LIN {X 0,Y 337.999,Z 716.277,A -85,B 0,C 180,E1 -25443.497,E2 -25443.497} C_VEL
LIN {X 0,Y 342.458,Z 719.963,A -85,B 0,C 180,E1 -25446.093,E2 -25446.093} C_VEL
LIN {X 0,Y 346.569,Z 722.702,A -85,B 0,C 180,E1 -25448.688,E2 -25448.688} C_VEL
LIN {X 0,Y 349.968,Z 724.791,A -85,B 0,C 180,E1 -25450.993,E2 -25450.993} C_VEL
LIN {X 0,Y 353.266,Z 727.665,A -85,B 0,C 180,E1 -25453.67,E2 -25453.67} C_VEL
LIN {X 0,Y 355.856,Z 729.583,A -85,B 0,C 180,E1 -25456.067,E2 -25456.067} C_VEL
LIN {X 0,Y 358.314,Z 731.084,A -85,B 0,C 180,E1 -25458.723,E2 -25458.723} C_VEL
LIN {X 0,Y 360.355,Z 731.966,A -85,B 0,C 180,E1 -25461.416,E2 -25461.416} C_VEL
LIN {X 0,Y 361.794,Z 732.692,A -85,B 0,C 180,E1 -25464.054,E2 -25464.054} C_VEL
LIN {X 0,Y 362.724,Z 733.17,A -85,B 0,C 180,E1 -25466.668,E2 -25466.668} C_VEL
LIN {X 0,Y 363.106,Z 733.308,A -85,B 0,C 180,E1 -25468.891,E2 -25468.891} C_VEL
LIN {X 0,Y 363.106,Z 733.292,A -85,B 0,C 180,E1 -25471.109,E2 -25471.109} C_VEL
LIN {X 0,Y 362.712,Z 733.195,A -85,B 0,C 180,E1 -25473.332,E2 -25473.332} C_VEL
LIN {X 0,Y 361.809,Z 732.656,A -85,B 0,C 180,E1 -25475.946,E2 -25475.946} C_VEL
LIN {X 0,Y 360.322,Z 731.939,A -85,B 0,C 180,E1 -25478.61,E2 -25478.61} C_VEL
LIN {X 0,Y 358.3,Z 731.072,A -85,B 0,C 180,E1 -25481.312,E2 -25481.312} C_VEL
LIN {X 0,Y 355.654,Z 729.459,A -85,B 0,C 180,E1 -25484.125,E2 -25484.125} C_VEL
LIN {X 0,Y 352.777,Z 727.309,A -85,B 0,C 180,E1 -25486.738,E2 -25486.738} C_VEL
LIN {X 0,Y 349.188,Z 724.198,A -85,B 0,C 180,E1 -25489.587,E2 -25489.587} C_VEL
LIN {X 0,Y 344.756,Z 721.495,A -85,B 0,C 180,E1 -25492.513,E2 -25492.513} C_VEL
LIN {X 0,Y 340.447,Z 718.436,A -85,B 0,C 180,E1 -25495.072,E2 -25495.072} C_VEL
LIN {X 0,Y 336.743,Z 715.339,A -85,B 0,C 180,E1 -25497.172,E2 -25497.172} C_VEL
LIN {X 0,Y 332.718,Z 712.68,A -85,B 0,C 180,E1 -25499.253,E2 -25499.253} C_VEL
LIN {X 0,Y 327.18,Z 708.25,A -85,B 0,C 180,E1 -25501.98,E2 -25501.98} C_VEL
LIN {X 0,Y 322.544,Z 704.803,A -85,B 0,C 180,E1 -25504.108,E2 -25504.108} C_VEL
LIN {X 0,Y 316.501,Z 699.903,A -85,B 0,C 180,E1 -25506.755,E2 -25506.755} C_VEL
LIN {X 0,Y 309.747,Z 694.783,A -85,B 0,C 180,E1 -25509.517,E2 -25509.517} C_VEL
LIN {X 0,Y 303.112,Z 689.395,A -85,B 0,C 180,E1 -25512.103,E2 -25512.103} C_VEL
LIN {X 0,Y 296.74,Z 684.407,A -85,B 0,C 180,E1 -25514.411,E2 -25514.411} C_VEL
LIN {X 0,Y 289.825,Z 679.065,A -85,B 0,C 180,E1 -25516.73,E2 -25516.73} C_VEL
LIN {X 0,Y 282.712,Z 673.492,A -85,B 0,C 180,E1 -25518.913,E2 -25518.913} C_VEL
LIN {X 0,Y 268.912,Z 662.781,A -85,B 0,C 180,E1 -25522.994,E2 -25522.994} C_VEL
LIN {X 0,Y 252.75,Z 647.426,A -85,B 0,C 180,E1 -25529.042,E2 -25529.042} C_VEL
LIN {X 0,Y 243.109,Z 634.604,A -85,B 0,C 180,E1 -25533.946,E2 -25533.946} C_VEL
LIN {X 0,Y 236.411,Z 622.152,A -85,B 0,C 180,E1 -25538.53,E2 -25538.53} C_VEL
LIN {X 0,Y 233.122,Z 614.521,A -85,B 0,C 180,E1 -25541.432,E2 -25541.432} C_VEL
LIN {X 0,Y 229.896,Z 607.668,A -85,B 0,C 180,E1 -25544.826,E2 -25544.826} C_VEL
LIN {X 0,Y 227.317,Z 602.559,A -85,B 0,C 180,E1 -25548.255,E2 -25548.255} C_VEL
LIN {X 0,Y 225.85,Z 599.593,A -85,B 0,C 180,E1 -25550.824,E2 -25550.824} C_VEL
LIN {X 0,Y 224.425,Z 596.183,A -85,B 0,C 180,E1 -25554.61,E2 -25554.61} C_VEL
LIN {X 0,Y 223.643,Z 595.09,A -85,B 0,C 180,E1 -25560,E2 -25560} C_VEL
LIN {X 0,Y 224.47,Z 596.375,A -85,B 0,C 180,E1 -25565.165,E2 -25565.165} C_VEL
LIN {X 0,Y 226.423,Z 600.662,A -85,B 0,C 180,E1 -25569.83,E2 -25569.83} C_VEL
LIN {X 0,Y 228.163,Z 604.251,A -85,B 0,C 180,E1 -25572.565,E2 -25572.565} C_VEL
LIN {X 0,Y 230.141,Z 608.221,A -85,B 0,C 180,E1 -25575.05,E2 -25575.05} C_VEL
LIN {X 0,Y 232.646,Z 613.57,A -85,B 0,C 180,E1 -25577.702,E2 -25577.702} C_VEL
LIN {X 0,Y 234.172,Z 617.919,A -85,B 0,C 180,E1 -25579.22,E2 -25579.22} C_VEL
LIN {X 0,Y 228.253,Z 677.793,A -85,B 0,C 180,E1 -25580.525,E2 -25580.525} C_VEL
LIN {X 0,Y 225.904,Z 694.176,A -85,B 0,C 180,E1 -25580.947,E2 -25580.947} C_VEL
LIN {X 0,Y 222.958,Z 708.344,A -85,B 0,C 180,E1 -25581.432,E2 -25581.432} C_VEL
LIN {X 0,Y 219.343,Z 721.676,A -85,B 0,C 180,E1 -25582.002,E2 -25582.002} C_VEL
LIN {X 0,Y 215.576,Z 733.24,A -85,B 0,C 180,E1 -25582.632,E2 -25582.632} C_VEL
LIN {X 0,Y 210.564,Z 746.285,A -85,B 0,C 180,E1 -25583.53,E2 -25583.53} C_VEL
LIN {X 0,Y 204.879,Z 759,A -85,B 0,C 180,E1 -25584.631,E2 -25584.631} C_VEL
LIN {X 0,Y 199.091,Z 770.319,A -85,B 0,C 180,E1 -25585.824,E2 -25585.824} C_VEL
LIN {X 0,Y 192.723,Z 781.446,A -85,B 0,C 180,E1 -25587.27,E2 -25587.27} C_VEL
LIN {X 0,Y 185.768,Z 792.275,A -85,B 0,C 180,E1 -25588.973,E2 -25588.973} C_VEL
LIN {X 0,Y 179.725,Z 800.954,A -85,B 0,C 180,E1 -25590.653,E2 -25590.653} C_VEL
LIN {X 0,Y 173.216,Z 809.59,A -85,B 0,C 180,E1 -25592.661,E2 -25592.661} C_VEL
LIN {X 0,Y 164.386,Z 820.104,A -85,B 0,C 180,E1 -25595.68,E2 -25595.68} C_VEL
LIN {X 0,Y 157.519,Z 827.783,A -85,B 0,C 180,E1 -25598.491,E2 -25598.491} C_VEL
LIN {X 0,Y 150.758,Z 834.958,A -85,B 0,C 180,E1 -25601.766,E2 -25601.766} C_VEL
LIN {X 0,Y 144.568,Z 841.096,A -85,B 0,C 180,E1 -25605.18,E2 -25605.18} C_VEL
LIN {X 0,Y 137.225,Z 848.046,A -85,B 0,C 180,E1 -25610.195,E2 -25610.195} C_VEL
LIN {X 0,Y 131.064,Z 853.813,A -85,B 0,C 180,E1 -25615.735,E2 -25615.735} C_VEL
LIN {X 0,Y 127.275,Z 857.437,A -85,B 0,C 180,E1 -25620.201,E2 -25620.201} C_VEL
LIN {X 0,Y 123.381,Z 861.307,A -85,B 0,C 180,E1 -25626.502,E2 -25626.502} C_VEL
LIN {X 0,Y 120.659,Z 864.176,A -85,B 0,C 180,E1 -25633.069,E2 -25633.069} C_VEL
LIN {X 0,Y 119.367,Z 866.085,A -85,B 0,C 180,E1 -25639.827,E2 -25639.827} C_VEL
LIN {X 0,Y 119.17,Z 866.774,A -85,B 0,C 180,E1 -25643.226,E2 -25643.226} C_VEL
LIN {X 0,Y 119.331,Z 867.267,A -85,B 0,C 180,E1 -25650,E2 -25650} C_VEL
LIN {X 0,Y 119.17,Z 866.774,A -85,B 0,C 180,E1 -25656.774,E2 -25656.774} C_VEL
LIN {X 0,Y 119.854,Z 865.323,A -85,B 0,C 180,E1 -25663.565,E2 -25663.565} C_VEL
LIN {X 0,Y 121.851,Z 862.917,A -85,B 0,C 180,E1 -25670.246,E2 -25670.246} C_VEL
LIN {X 0,Y 125.192,Z 859.526,A -85,B 0,C 180,E1 -25676.685,E2 -25676.685} C_VEL
LIN {X 0,Y 129.705,Z 855.102,A -85,B 0,C 180,E1 -25682.808,E2 -25682.808} C_VEL
LIN {X 0,Y 135.589,Z 849.593,A -85,B 0,C 180,E1 -25688.461,E2 -25688.461} C_VEL
LIN {X 0,Y 140.755,Z 844.73,A -85,B 0,C 180,E1 -25692.38,E2 -25692.38} C_VEL
LIN {X 0,Y 146.39,Z 839.356,A -85,B 0,C 180,E1 -25695.871,E2 -25695.871} C_VEL
LIN {X 0,Y 148.823,Z 836.554,A -85,B 0,C 180,E1 -25697.657,E2 -25697.657} C_VEL
LIN {X 0,Y 151.551,Z 831.851,A -85,B 0,C 180,E1 -25700.824,E2 -25700.824} C_VEL
LIN {X 0,Y 154.515,Z 826.734,A -85,B 0,C 180,E1 -25703.808,E2 -25703.808} C_VEL
LIN {X 0,Y 157.216,Z 823.286,A -85,B 0,C 180,E1 -25705.266,E2 -25705.266} C_VEL
LIN {X 0,Y 165.406,Z 814.068,A -85,B 0,C 180,E1 -25708.186,E2 -25708.186} C_VEL
LIN {X 0,Y 173.438,Z 804.341,A -85,B 0,C 180,E1 -25710.565,E2 -25710.565} C_VEL
LIN {X 0,Y 180.924,Z 794.175,A -85,B 0,C 180,E1 -25712.632,E2 -25712.632} C_VEL
LIN {X 0,Y 188.08,Z 783.518,A -85,B 0,C 180,E1 -25714.351,E2 -25714.351} C_VEL
LIN {X 0,Y 194.601,Z 772.715,A -85,B 0,C 180,E1 -25715.766,E2 -25715.766} C_VEL
LIN {X 0,Y 200.524,Z 761.787,A -85,B 0,C 180,E1 -25716.925,E2 -25716.925} C_VEL
LIN {X 0,Y 206.343,Z 749.49,A -85,B 0,C 180,E1 -25718.009,E2 -25718.009} C_VEL
LIN {X 0,Y 211.426,Z 737.132,A -85,B 0,C 180,E1 -25718.876,E2 -25718.876} C_VEL
LIN {X 0,Y 215.627,Z 725.167,A -85,B 0,C 180,E1 -25719.56,E2 -25719.56} C_VEL
LIN {X 0,Y 219.498,Z 711.964,A -85,B 0,C 180,E1 -25720.139,E2 -25720.139} C_VEL
LIN {X 0,Y 222.58,Z 698.598,A -85,B 0,C 180,E1 -25720.611,E2 -25720.611} C_VEL
LIN {X 0,Y 224.742,Z 686.018,A -85,B 0,C 180,E1 -25720.968,E2 -25720.968} C_VEL
LIN {X 0,Y 228.136,Z 655.335,A -85,B 0,C 180,E1 -25721.627,E2 -25721.627} C_VEL
LIN {X 0,Y 231.565,Z 621.607,A -85,B 0,C 180,E1 -25722.332,E2 -25722.332} C_VEL
LIN {X 0,Y 229.974,Z 617.635,A -85,B 0,C 180,E1 -25724.035,E2 -25724.035} C_VEL
LIN {X 0,Y 227.684,Z 612.618,A -85,B 0,C 180,E1 -25726.813,E2 -25726.813} C_VEL
LIN {X 0,Y 225.971,Z 609.022,A -85,B 0,C 180,E1 -25729.358,E2 -25729.358} C_VEL
LIN {X 0,Y 224.74,Z 606.367,A -85,B 0,C 180,E1 -25731.684,E2 -25731.684} C_VEL
LIN {X 0,Y 223.406,Z 603.177,A -85,B 0,C 180,E1 -25735.489,E2 -25735.489} C_VEL
LIN {X 0,Y 222.78,Z 602.124,A -85,B 0,C 180,E1 -25740,E2 -25740} C_VEL
LIN {X 0,Y 223.536,Z 603.452,A -85,B 0,C 180,E1 -25745.412,E2 -25745.412} C_VEL
LIN {X 0,Y 225.251,Z 607.461,A -85,B 0,C 180,E1 -25749.767,E2 -25749.767} C_VEL
LIN {X 0,Y 226.899,Z 611.077,A -85,B 0,C 180,E1 -25752.522,E2 -25752.522} C_VEL
LIN {X 0,Y 229.124,Z 615.63,A -85,B 0,C 180,E1 -25755.397,E2 -25755.397} C_VEL
LIN {X 0,Y 232.457,Z 623.396,A -85,B 0,C 180,E1 -25758.923,E2 -25758.923} C_VEL
LIN {X 0,Y 239.806,Z 638.871,A -85,B 0,C 180,E1 -25764.678,E2 -25764.678} C_VEL
LIN {X 0,Y 246.178,Z 648.31,A -85,B 0,C 180,E1 -25768.334,E2 -25768.334} C_VEL
LIN {X 0,Y 253.816,Z 657.284,A -85,B 0,C 180,E1 -25771.884,E2 -25771.884} C_VEL
LIN {X 0,Y 270.22,Z 672.233,A -85,B 0,C 180,E1 -25777.803,E2 -25777.803} C_VEL
LIN {X 0,Y 281.302,Z 680.788,A -85,B 0,C 180,E1 -25781.1,E2 -25781.1} C_VEL
LIN {X 0,Y 289.149,Z 686.906,A -85,B 0,C 180,E1 -25783.564,E2 -25783.564} C_VEL
LIN {X 0,Y 295.479,Z 691.92,A -85,B 0,C 180,E1 -25785.734,E2 -25785.734} C_VEL
LIN {X 0,Y 302.486,Z 697.251,A -85,B 0,C 180,E1 -25788.279,E2 -25788.279} C_VEL
LIN {X 0,Y 309.232,Z 702.759,A -85,B 0,C 180,E1 -25790.927,E2 -25790.927} C_VEL
LIN {X 0,Y 315.134,Z 707.221,A -85,B 0,C 180,E1 -25793.337,E2 -25793.337} C_VEL
LIN {X 0,Y 321.273,Z 711.966,A -85,B 0,C 180,E1 -25796.008,E2 -25796.008} C_VEL
LIN {X 0,Y 325.921,Z 715.518,A -85,B 0,C 180,E1 -25798.147,E2 -25798.147} C_VEL
LIN {X 0,Y 330.655,Z 719.336,A -85,B 0,C 180,E1 -25800.489,E2 -25800.489} C_VEL
LIN {X 0,Y 336.004,Z 722.897,A -85,B 0,C 180,E1 -25803.223,E2 -25803.223} C_VEL
LIN {X 0,Y 340.681,Z 726.787,A -85,B 0,C 180,E1 -25805.96,E2 -25805.96} C_VEL
LIN {X 0,Y 344.422,Z 729.295,A -85,B 0,C 180,E1 -25808.279,E2 -25808.279} C_VEL
LIN {X 0,Y 348.222,Z 731.574,A -85,B 0,C 180,E1 -25810.811,E2 -25810.811} C_VEL
LIN {X 0,Y 351.453,Z 734.418,A -85,B 0,C 180,E1 -25813.424,E2 -25813.424} C_VEL
LIN {X 0,Y 354.249,Z 736.481,A -85,B 0,C 180,E1 -25815.986,E2 -25815.986} C_VEL
LIN {X 0,Y 356.766,Z 737.985,A -85,B 0,C 180,E1 -25818.639,E2 -25818.639} C_VEL
LIN {X 0,Y 358.867,Z 738.904,A -85,B 0,C 180,E1 -25821.38,E2 -25821.38} C_VEL
LIN {X 0,Y 360.357,Z 739.625,A -85,B 0,C 180,E1 -25824.063,E2 -25824.063} C_VEL
LIN {X 0,Y 361.291,Z 740.1,A -85,B 0,C 180,E1 -25826.655,E2 -25826.655} C_VEL
LIN {X 0,Y 361.676,Z 740.233,A -85,B 0,C 180,E1 -25828.887,E2 -25828.887} C_VEL
LIN {X 0,Y 361.666,Z 740.244,A -85,B 0,C 180,E1 -25831.113,E2 -25831.113} C_VEL
LIN {X 0,Y 361.262,Z 740.134,A -85,B 0,C 180,E1 -25833.346,E2 -25833.346} C_VEL
LIN {X 0,Y 360.371,Z 739.604,A -85,B 0,C 180,E1 -25835.959,E2 -25835.959} C_VEL
LIN {X 0,Y 358.852,Z 738.88,A -85,B 0,C 180,E1 -25838.646,E2 -25838.646} C_VEL
LIN {X 0,Y 356.756,Z 737.994,A -85,B 0,C 180,E1 -25841.361,E2 -25841.361} C_VEL
LIN {X 0,Y 354.243,Z 736.464,A -85,B 0,C 180,E1 -25844.021,E2 -25844.021} C_VEL
LIN {X 0,Y 351.154,Z 734.21,A -85,B 0,C 180,E1 -25846.818,E2 -25846.818} C_VEL
LIN {X 0,Y 347.641,Z 731.128,A -85,B 0,C 180,E1 -25849.603,E2 -25849.603} C_VEL
LIN {X 0,Y 343.959,Z 728.983,A -85,B 0,C 180,E1 -25852.019,E2 -25852.019} C_VEL
LIN {X 0,Y 340.235,Z 726.499,A -85,B 0,C 180,E1 -25854.291,E2 -25854.291} C_VEL
LIN {X 0,Y 335.631,Z 722.524,A -85,B 0,C 180,E1 -25856.993,E2 -25856.993} C_VEL
LIN {X 0,Y 330.992,Z 719.572,A -85,B 0,C 180,E1 -25859.344,E2 -25859.344} C_VEL
LIN {X 0,Y 325.589,Z 715.32,A -85,B 0,C 180,E1 -25861.996,E2 -25861.996} C_VEL
LIN {X 0,Y 322.005,Z 712.477,A -85,B 0,C 180,E1 -25863.666,E2 -25863.666} C_VEL
LIN {X 0,Y 315.88,Z 707.869,A -85,B 0,C 180,E1 -25866.331,E2 -25866.331} C_VEL
LIN {X 0,Y 310.932,Z 703.991,A -85,B 0,C 180,E1 -25868.4,E2 -25868.4} C_VEL
LIN {X 0,Y 304.177,Z 698.648,A -85,B 0,C 180,E1 -25871.074,E2 -25871.074} C_VEL
LIN {X 0,Y 296.872,Z 693.051,A -85,B 0,C 180,E1 -25873.772,E2 -25873.772} C_VEL
LIN {X 0,Y 290.435,Z 687.889,A -85,B 0,C 180,E1 -25876.007,E2 -25876.007} C_VEL
LIN {X 0,Y 283.045,Z 682.12,A -85,B 0,C 180,E1 -25878.38,E2 -25878.38} C_VEL
LIN {X 0,Y 273.692,Z 674.999,A -85,B 0,C 180,E1 -25881.126,E2 -25881.126} C_VEL
LIN {X 0,Y 255.909,Z 659.417,A -85,B 0,C 180,E1 -25887.256,E2 -25887.256} C_VEL
LIN {X 0,Y 247.388,Z 649.9,A -85,B 0,C 180,E1 -25891.052,E2 -25891.052} C_VEL
LIN {X 0,Y 240.504,Z 640.005,A -85,B 0,C 180,E1 -25894.88,E2 -25894.88} C_VEL
LIN {X 0,Y 234.442,Z 628.281,A -85,B 0,C 180,E1 -25899.272,E2 -25899.272} C_VEL
LIN {X 0,Y 231.273,Z 620.562,A -85,B 0,C 180,E1 -25902.247,E2 -25902.247} C_VEL
LIN {X 0,Y 228.281,Z 613.826,A -85,B 0,C 180,E1 -25905.628,E2 -25905.628} C_VEL
LIN {X 0,Y 226.014,Z 609.158,A -85,B 0,C 180,E1 -25908.862,E2 -25908.862} C_VEL
LIN {X 0,Y 224.752,Z 606.438,A -85,B 0,C 180,E1 -25911.232,E2 -25911.232} C_VEL
LIN {X 0,Y 223.395,Z 603.106,A -85,B 0,C 180,E1 -25915.136,E2 -25915.136} C_VEL
LIN {X 0,Y 222.777,Z 602.147,A -85,B 0,C 180,E1 -25920,E2 -25920} C_VEL
LIN {X 0,Y 223.527,Z 603.424,A -85,B 0,C 180,E1 -25924.961,E2 -25924.961} C_VEL
LIN {X 0,Y 225.239,Z 607.366,A -85,B 0,C 180,E1 -25929.315,E2 -25929.315} C_VEL
LIN {X 0,Y 226.88,Z 610.976,A -85,B 0,C 180,E1 -25932.069,E2 -25932.069} C_VEL
LIN {X 0,Y 229.06,Z 615.498,A -85,B 0,C 180,E1 -25934.907,E2 -25934.907} C_VEL
LIN {X 0,Y 231.421,Z 621.118,A -85,B 0,C 180,E1 -25937.508,E2 -25937.508} C_VEL
LIN {X 0,Y 231.564,Z 621.621,A -85,B 0,C 180,E1 -25937.668,E2 -25937.668} C_VEL
LIN {X 0,Y 224.979,Z 684.568,A -85,B 0,C 180,E1 -25939.01,E2 -25939.01} C_VEL
LIN {X 0,Y 222.386,Z 699.597,A -85,B 0,C 180,E1 -25939.418,E2 -25939.418} C_VEL
LIN {X 0,Y 218.329,Z 716.503,A -85,B 0,C 180,E1 -25940.029,E2 -25940.029} C_VEL
LIN {X 0,Y 212.933,Z 733.029,A -85,B 0,C 180,E1 -25940.861,E2 -25940.861} C_VEL
LIN {X 0,Y 207.7,Z 746.354,A -85,B 0,C 180,E1 -25941.75,E2 -25941.75} C_VEL
LIN {X 0,Y 202.009,Z 758.789,A -85,B 0,C 180,E1 -25942.791,E2 -25942.791} C_VEL
LIN {X 0,Y 196.091,Z 770.109,A -85,B 0,C 180,E1 -25943.949,E2 -25943.949} C_VEL
LIN {X 0,Y 189.552,Z 781.234,A -85,B 0,C 180,E1 -25945.348,E2 -25945.348} C_VEL
LIN {X 0,Y 182.386,Z 792.062,A -85,B 0,C 180,E1 -25946.992,E2 -25946.992} C_VEL
LIN {X 0,Y 176.18,Z 800.742,A -85,B 0,C 180,E1 -25948.648,E2 -25948.648} C_VEL
LIN {X 0,Y 168.104,Z 810.942,A -85,B 0,C 180,E1 -25951.015,E2 -25951.015} C_VEL
LIN {X 0,Y 160.315,Z 819.892,A -85,B 0,C 180,E1 -25953.6,E2 -25953.6} C_VEL
LIN {X 0,Y 152.929,Z 827.782,A -85,B 0,C 180,E1 -25956.468,E2 -25956.468} C_VEL
LIN {X 0,Y 146.036,Z 834.745,A -85,B 0,C 180,E1 -25959.647,E2 -25959.647} C_VEL
LIN {X 0,Y 139.535,Z 840.883,A -85,B 0,C 180,E1 -25963.088,E2 -25963.088} C_VEL
LIN {X 0,Y 133.61,Z 846.287,A -85,B 0,C 180,E1 -25966.859,E2 -25966.859} C_VEL
LIN {X 0,Y 126.709,Z 852.311,A -85,B 0,C 180,E1 -25972.403,E2 -25972.403} C_VEL
LIN {X 0,Y 121.044,Z 857.223,A -85,B 0,C 180,E1 -25978.497,E2 -25978.497} C_VEL
LIN {X 0,Y 116.805,Z 861.094,A -85,B 0,C 180,E1 -25985.091,E2 -25985.091} C_VEL
LIN {X 0,Y 113.824,Z 863.964,A -85,B 0,C 180,E1 -25992.018,E2 -25992.018} C_VEL
LIN {X 0,Y 112.348,Z 865.874,A -85,B 0,C 180,E1 -25999.184,E2 -25999.184} C_VEL
LIN {X 0,Y 112.091,Z 866.563,A -85,B 0,C 180,E1 -26002.796,E2 -26002.796} C_VEL
LIN {X 0,Y 112.248,Z 867.057,A -85,B 0,C 180,E1 -26010,E2 -26010} C_VEL
LIN {X 0,Y 112.091,Z 866.563,A -85,B 0,C 180,E1 -26017.204,E2 -26017.204} C_VEL
LIN {X 0,Y 112.883,Z 865.111,A -85,B 0,C 180,E1 -26024.42,E2 -26024.42} C_VEL
LIN {X 0,Y 115.125,Z 862.704,A -85,B 0,C 180,E1 -26031.486,E2 -26031.486} C_VEL
LIN {X 0,Y 118.79,Z 859.313,A -85,B 0,C 180,E1 -26038.248,E2 -26038.248} C_VEL
LIN {X 0,Y 123.691,Z 854.889,A -85,B 0,C 180,E1 -26044.623,E2 -26044.623} C_VEL
LIN {X 0,Y 129.997,Z 849.379,A -85,B 0,C 180,E1 -26050.447,E2 -26050.447} C_VEL
LIN {X 0,Y 135.517,Z 844.517,A -85,B 0,C 180,E1 -26054.435,E2 -26054.435} C_VEL
LIN {X 0,Y 143.851,Z 836.851,A -85,B 0,C 180,E1 -26059.222,E2 -26059.222} C_VEL
LIN {X 0,Y 150.581,Z 830.197,A -85,B 0,C 180,E1 -26062.506,E2 -26062.506} C_VEL
LIN {X 0,Y 157.216,Z 823.286,A -85,B 0,C 180,E1 -26065.266,E2 -26065.266} C_VEL
LIN {X 0,Y 160.007,Z 819.792,A -85,B 0,C 180,E1 -26066.647,E2 -26066.647} C_VEL
LIN {X 0,Y 167.271,Z 808.009,A -85,B 0,C 180,E1 -26071.607,E2 -26071.607} C_VEL
LIN {X 0,Y 170.147,Z 803.963,A -85,B 0,C 180,E1 -26072.713,E2 -26072.713} C_VEL
LIN {X 0,Y 178.527,Z 792.857,A -85,B 0,C 180,E1 -26074.878,E2 -26074.878} C_VEL
LIN {X 0,Y 185.105,Z 783.307,A -85,B 0,C 180,E1 -26076.341,E2 -26076.341} C_VEL
LIN {X 0,Y 191.789,Z 772.505,A -85,B 0,C 180,E1 -26077.706,E2 -26077.706} C_VEL
LIN {X 0,Y 197.741,Z 761.767,A -85,B 0,C 180,E1 -26078.808,E2 -26078.808} C_VEL
LIN {X 0,Y 203.782,Z 749.279,A -85,B 0,C 180,E1 -26079.868,E2 -26079.868} C_VEL
LIN {X 0,Y 208.963,Z 736.921,A -85,B 0,C 180,E1 -26080.699,E2 -26080.699} C_VEL
LIN {X 0,Y 213.247,Z 724.957,A -85,B 0,C 180,E1 -26081.351,E2 -26081.351} C_VEL
LIN {X 0,Y 217.191,Z 711.754,A -85,B 0,C 180,E1 -26081.899,E2 -26081.899} C_VEL
LIN {X 0,Y 220.323,Z 698.388,A -85,B 0,C 180,E1 -26082.354,E2 -26082.354} C_VEL
LIN {X 0,Y 222.443,Z 686.442,A -85,B 0,C 180,E1 -26082.682,E2 -26082.682} C_VEL
LIN {X 0,Y 225.705,Z 657.977,A -85,B 0,C 180,E1 -26083.275,E2 -26083.275} C_VEL
LIN {X 0,Y 229.068,Z 625.66,A -85,B 0,C 180,E1 -26083.933,E2 -26083.933} C_VEL
LIN {X 0,Y 226.998,Z 620.729,A -85,B 0,C 180,E1 -26086.459,E2 -26086.459} C_VEL
LIN {X 0,Y 224.822,Z 615.841,A -85,B 0,C 180,E1 -26089.758,E2 -26089.758} C_VEL
LIN {X 0,Y 223.706,Z 613.291,A -85,B 0,C 180,E1 -26091.986,E2 -26091.986} C_VEL
LIN {X 0,Y 222.543,Z 610.231,A -85,B 0,C 180,E1 -26095.471,E2 -26095.471} C_VEL
LIN {X 0,Y 221.914,Z 609.176,A -85,B 0,C 180,E1 -26100,E2 -26100} C_VEL
LIN {X 0,Y 222.556,Z 610.306,A -85,B 0,C 180,E1 -26105.015,E2 -26105.015} C_VEL
LIN {X 0,Y 224.138,Z 614.289,A -85,B 0,C 180,E1 -26109.361,E2 -26109.361} C_VEL
LIN {X 0,Y 225.658,Z 617.814,A -85,B 0,C 180,E1 -26112.055,E2 -26112.055} C_VEL
LIN {X 0,Y 227.629,Z 622.06,A -85,B 0,C 180,E1 -26114.756,E2 -26114.756} C_VEL
LIN {X 0,Y 230.625,Z 629.493,A -85,B 0,C 180,E1 -26118.143,E2 -26118.143} C_VEL
LIN {X 0,Y 237.705,Z 645.024,A -85,B 0,C 180,E1 -26123.996,E2 -26123.996} C_VEL
LIN {X 0,Y 243.985,Z 654.581,A -85,B 0,C 180,E1 -26127.749,E2 -26127.749} C_VEL
LIN {X 0,Y 251.575,Z 663.663,A -85,B 0,C 180,E1 -26131.393,E2 -26131.393} C_VEL
LIN {X 0,Y 267.106,Z 678.173,A -85,B 0,C 180,E1 -26137.24,E2 -26137.24} C_VEL
LIN {X 0,Y 281.406,Z 689.419,A -85,B 0,C 180,E1 -26141.678,E2 -26141.678} C_VEL
LIN {X 0,Y 289.178,Z 695.327,A -85,B 0,C 180,E1 -26144.202,E2 -26144.202} C_VEL
LIN {X 0,Y 296.503,Z 701.217,A -85,B 0,C 180,E1 -26146.783,E2 -26146.783} C_VEL
LIN {X 0,Y 303.158,Z 706.395,A -85,B 0,C 180,E1 -26149.27,E2 -26149.27} C_VEL
LIN {X 0,Y 309.384,Z 711.179,A -85,B 0,C 180,E1 -26151.739,E2 -26151.739} C_VEL
LIN {X 0,Y 314.444,Z 715.198,A -85,B 0,C 180,E1 -26153.846,E2 -26153.846} C_VEL
LIN {X 0,Y 320.403,Z 719.619,A -85,B 0,C 180,E1 -26156.462,E2 -26156.462} C_VEL
LIN {X 0,Y 324.538,Z 722.952,A -85,B 0,C 180,E1 -26158.392,E2 -26158.392} C_VEL
LIN {X 0,Y 329.924,Z 727.044,A -85,B 0,C 180,E1 -26161.033,E2 -26161.033} C_VEL
LIN {X 0,Y 334.237,Z 729.895,A -85,B 0,C 180,E1 -26163.272,E2 -26163.272} C_VEL
LIN {X 0,Y 338.14,Z 733.169,A -85,B 0,C 180,E1 -26165.549,E2 -26165.549} C_VEL
LIN {X 0,Y 342.242,Z 735.939,A -85,B 0,C 180,E1 -26168.047,E2 -26168.047} C_VEL
LIN {X 0,Y 346.31,Z 738.405,A -85,B 0,C 180,E1 -26170.724,E2 -26170.724} C_VEL
LIN {X 0,Y 349.713,Z 741.37,A -85,B 0,C 180,E1 -26173.504,E2 -26173.504} C_VEL
LIN {X 0,Y 352.619,Z 743.467,A -85,B 0,C 180,E1 -26176.163,E2 -26176.163} C_VEL
LIN {X 0,Y 354.89,Z 744.81,A -85,B 0,C 180,E1 -26178.578,E2 -26178.578} C_VEL
LIN {X 0,Y 357.041,Z 745.751,A -85,B 0,C 180,E1 -26181.335,E2 -26181.335} C_VEL
LIN {X 0,Y 358.585,Z 746.488,A -85,B 0,C 180,E1 -26184.033,E2 -26184.033} C_VEL
LIN {X 0,Y 359.539,Z 746.952,A -85,B 0,C 180,E1 -26186.638,E2 -26186.638} C_VEL
LIN {X 0,Y 359.93,Z 747.092,A -85,B 0,C 180,E1 -26188.881,E2 -26188.881} C_VEL
LIN {X 0,Y 359.917,Z 747.097,A -85,B 0,C 180,E1 -26191.119,E2 -26191.119} C_VEL
LIN {X 0,Y 359.502,Z 746.994,A -85,B 0,C 180,E1 -26193.362,E2 -26193.362} C_VEL
LIN {X 0,Y 358.59,Z 746.47,A -85,B 0,C 180,E1 -26195.989,E2 -26195.989} C_VEL
LIN {X 0,Y 357.032,Z 745.737,A -85,B 0,C 180,E1 -26198.69,E2 -26198.69} C_VEL
LIN {X 0,Y 354.865,Z 744.808,A -85,B 0,C 180,E1 -26201.423,E2 -26201.423} C_VEL
LIN {X 0,Y 352.356,Z 743.28,A -85,B 0,C 180,E1 -26204.098,E2 -26204.098} C_VEL
LIN {X 0,Y 349.375,Z 741.116,A -85,B 0,C 180,E1 -26206.781,E2 -26206.781} C_VEL
LIN {X 0,Y 346.087,Z 738.144,A -85,B 0,C 180,E1 -26209.458,E2 -26209.458} C_VEL
LIN {X 0,Y 342.128,Z 735.828,A -85,B 0,C 180,E1 -26212.032,E2 -26212.032} C_VEL
LIN {X 0,Y 338.051,Z 733.143,A -85,B 0,C 180,E1 -26214.498,E2 -26214.498} C_VEL
LIN {X 0,Y 334.149,Z 729.856,A -85,B 0,C 180,E1 -26216.758,E2 -26216.758} C_VEL
LIN {X 0,Y 328.848,Z 726.245,A -85,B 0,C 180,E1 -26219.518,E2 -26219.518} C_VEL
LIN {X 0,Y 323.237,Z 721.879,A -85,B 0,C 180,E1 -26222.225,E2 -26222.225} C_VEL
LIN {X 0,Y 319.653,Z 719.093,A -85,B 0,C 180,E1 -26223.867,E2 -26223.867} C_VEL
LIN {X 0,Y 313.69,Z 714.596,A -85,B 0,C 180,E1 -26226.469,E2 -26226.469} C_VEL
LIN {X 0,Y 308.902,Z 710.843,A -85,B 0,C 180,E1 -26228.449,E2 -26228.449} C_VEL
LIN {X 0,Y 302.529,Z 705.917,A -85,B 0,C 180,E1 -26230.967,E2 -26230.967} C_VEL
LIN {X 0,Y 295.881,Z 700.724,A -85,B 0,C 180,E1 -26233.447,E2 -26233.447} C_VEL
LIN {X 0,Y 288.265,Z 694.65,A -85,B 0,C 180,E1 -26236.108,E2 -26236.108} C_VEL
LIN {X 0,Y 280.806,Z 688.913,A -85,B 0,C 180,E1 -26238.513,E2 -26238.513} C_VEL
LIN {X 0,Y 264.377,Z 675.876,A -85,B 0,C 180,E1 -26243.68,E2 -26243.68} C_VEL
LIN {X 0,Y 248.796,Z 660.704,A -85,B 0,C 180,E1 -26249.848,E2 -26249.848} C_VEL
LIN {X 0,Y 238.885,Z 647.079,A -85,B 0,C 180,E1 -26255.224,E2 -26255.224} C_VEL
LIN {X 0,Y 232.24,Z 633.708,A -85,B 0,C 180,E1 -26260.278,E2 -26260.278} C_VEL
LIN {X 0,Y 229.527,Z 626.721,A -85,B 0,C 180,E1 -26263.016,E2 -26263.016} C_VEL
LIN {X 0,Y 226.773,Z 620.104,A -85,B 0,C 180,E1 -26266.36,E2 -26266.36} C_VEL
LIN {X 0,Y 224.652,Z 615.521,A -85,B 0,C 180,E1 -26269.638,E2 -26269.638} C_VEL
LIN {X 0,Y 223.692,Z 613.321,A -85,B 0,C 180,E1 -26271.588,E2 -26271.588} C_VEL
LIN {X 0,Y 222.528,Z 610.188,A -85,B 0,C 180,E1 -26275.117,E2 -26275.117} C_VEL
LIN {X 0,Y 221.911,Z 609.2,A -85,B 0,C 180,E1 -26280,E2 -26280} C_VEL
LIN {X 0,Y 222.564,Z 610.358,A -85,B 0,C 180,E1 -26284.642,E2 -26284.642} C_VEL
LIN {X 0,Y 224.175,Z 614.369,A -85,B 0,C 180,E1 -26289.019,E2 -26289.019} C_VEL
LIN {X 0,Y 225.566,Z 617.546,A -85,B 0,C 180,E1 -26291.485,E2 -26291.485} C_VEL
LIN {X 0,Y 227.639,Z 622.115,A -85,B 0,C 180,E1 -26294.357,E2 -26294.357} C_VEL
LIN {X 0,Y 229.071,Z 625.664,A -85,B 0,C 180,E1 -26296.071,E2 -26296.071} C_VEL
LIN {X 0,Y 222.83,Z 683.844,A -85,B 0,C 180,E1 -26297.261,E2 -26297.261} C_VEL
LIN {X 0,Y 220.325,Z 698.388,A -85,B 0,C 180,E1 -26297.647,E2 -26297.647} C_VEL
LIN {X 0,Y 216.985,Z 712.519,A -85,B 0,C 180,E1 -26298.121,E2 -26298.121} C_VEL
LIN {X 0,Y 211.674,Z 729.743,A -85,B 0,C 180,E1 -26298.874,E2 -26298.874} C_VEL
LIN {X 0,Y 205.467,Z 745.454,A -85,B 0,C 180,E1 -26299.848,E2 -26299.848} C_VEL
LIN {X 0,Y 199.97,Z 757.387,A -85,B 0,C 180,E1 -26300.801,E2 -26300.801} C_VEL
LIN {X 0,Y 193.307,Z 769.898,A -85,B 0,C 180,E1 -26302.017,E2 -26302.017} C_VEL
LIN {X 0,Y 186.595,Z 781.022,A -85,B 0,C 180,E1 -26303.357,E2 -26303.357} C_VEL
LIN {X 0,Y 179.249,Z 791.851,A -85,B 0,C 180,E1 -26304.952,E2 -26304.952} C_VEL
LIN {X 0,Y 171.594,Z 802.11,A -85,B 0,C 180,E1 -26306.885,E2 -26306.885} C_VEL
LIN {X 0,Y 164.532,Z 810.731,A -85,B 0,C 180,E1 -26308.879,E2 -26308.879} C_VEL
LIN {X 0,Y 156.445,Z 819.68,A -85,B 0,C 180,E1 -26311.403,E2 -26311.403} C_VEL
LIN {X 0,Y 148.766,Z 827.569,A -85,B 0,C 180,E1 -26314.24,E2 -26314.24} C_VEL
LIN {X 0,Y 141.537,Z 834.531,A -85,B 0,C 180,E1 -26317.396,E2 -26317.396} C_VEL
LIN {X 0,Y 134.717,Z 840.67,A -85,B 0,C 180,E1 -26320.85,E2 -26320.85} C_VEL
LIN {X 0,Y 126.595,Z 847.523,A -85,B 0,C 180,E1 -26325.92,E2 -26325.92} C_VEL
LIN {X 0,Y 119.414,Z 853.387,A -85,B 0,C 180,E1 -26331.833,E2 -26331.833} C_VEL
LIN {X 0,Y 114.951,Z 857.01,A -85,B 0,C 180,E1 -26336.617,E2 -26336.617} C_VEL
LIN {X 0,Y 110.31,Z 860.881,A -85,B 0,C 180,E1 -26343.515,E2 -26343.515} C_VEL
LIN {X 0,Y 107.033,Z 863.752,A -85,B 0,C 180,E1 -26350.834,E2 -26350.834} C_VEL
LIN {X 0,Y 105.32,Z 865.662,A -85,B 0,C 180,E1 -26358.452,E2 -26358.452} C_VEL
LIN {X 0,Y 105.016,Z 866.352,A -85,B 0,C 180,E1 -26362.308,E2 -26362.308} C_VEL
LIN {X 0,Y 105.166,Z 866.848,A -85,B 0,C 180,E1 -26370,E2 -26370} C_VEL
LIN {X 0,Y 105.016,Z 866.352,A -85,B 0,C 180,E1 -26377.692,E2 -26377.692} C_VEL
LIN {X 0,Y 105.944,Z 864.899,A -85,B 0,C 180,E1 -26385.387,E2 -26385.387} C_VEL
LIN {X 0,Y 108.461,Z 862.491,A -85,B 0,C 180,E1 -26392.878,E2 -26392.878} C_VEL
LIN {X 0,Y 112.46,Z 859.099,A -85,B 0,C 180,E1 -26399.996,E2 -26399.996} C_VEL
LIN {X 0,Y 117.815,Z 854.675,A -85,B 0,C 180,E1 -26406.621,E2 -26406.621} C_VEL
LIN {X 0,Y 124.577,Z 849.165,A -85,B 0,C 180,E1 -26412.607,E2 -26412.607} C_VEL
LIN {X 0,Y 130.462,Z 844.303,A -85,B 0,C 180,E1 -26416.655,E2 -26416.655} C_VEL
LIN {X 0,Y 139.245,Z 836.638,A -85,B 0,C 180,E1 -26421.472,E2 -26421.472} C_VEL
LIN {X 0,Y 146.532,Z 829.738,A -85,B 0,C 180,E1 -26424.862,E2 -26424.862} C_VEL
LIN {X 0,Y 153.816,Z 822.434,A -85,B 0,C 180,E1 -26427.7,E2 -26427.7} C_VEL
LIN {X 0,Y 161.731,Z 813.856,A -85,B 0,C 180,E1 -26430.351,E2 -26430.351} C_VEL
LIN {X 0,Y 170.147,Z 803.963,A -85,B 0,C 180,E1 -26432.713,E2 -26432.713} C_VEL
LIN {X 0,Y 171.917,Z 801.3,A -85,B 0,C 180,E1 -26433.497,E2 -26433.497} C_VEL
LIN {X 0,Y 175.7,Z 792.914,A -85,B 0,C 180,E1 -26436.764,E2 -26436.764} C_VEL
LIN {X 0,Y 177.586,Z 789.988,A -85,B 0,C 180,E1 -26437.411,E2 -26437.411} C_VEL
LIN {X 0,Y 186.89,Z 776.198,A -85,B 0,C 180,E1 -26439.293,E2 -26439.293} C_VEL
LIN {X 0,Y 195.175,Z 761.758,A -85,B 0,C 180,E1 -26440.74,E2 -26440.74} C_VEL
LIN {X 0,Y 201.44,Z 749.069,A -85,B 0,C 180,E1 -26441.771,E2 -26441.771} C_VEL
LIN {X 0,Y 206.716,Z 736.711,A -85,B 0,C 180,E1 -26442.565,E2 -26442.565} C_VEL
LIN {X 0,Y 211.086,Z 724.748,A -85,B 0,C 180,E1 -26443.175,E2 -26443.175} C_VEL
LIN {X 0,Y 215.086,Z 711.544,A -85,B 0,C 180,E1 -26443.701,E2 -26443.701} C_VEL
LIN {X 0,Y 218.274,Z 698.178,A -85,B 0,C 180,E1 -26444.132,E2 -26444.132} C_VEL
LIN {X 0,Y 220.535,Z 685.41,A -85,B 0,C 180,E1 -26444.473,E2 -26444.473} C_VEL
LIN {X 0,Y 224.039,Z 655.16,A -85,B 0,C 180,E1 -26445.071,E2 -26445.071} C_VEL
LIN {X 0,Y 226.704,Z 630.02,A -85,B 0,C 180,E1 -26445.577,E2 -26445.577} C_VEL
LIN {X 0,Y 224.787,Z 625.332,A -85,B 0,C 180,E1 -26448.274,E2 -26448.274} C_VEL
LIN {X 0,Y 223.394,Z 621.988,A -85,B 0,C 180,E1 -26450.721,E2 -26450.721} C_VEL
LIN {X 0,Y 222.582,Z 620.035,A -85,B 0,C 180,E1 -26452.516,E2 -26452.516} C_VEL
LIN {X 0,Y 221.552,Z 617.19,A -85,B 0,C 180,E1 -26455.907,E2 -26455.907} C_VEL
LIN {X 0,Y 221.048,Z 616.229,A -85,B 0,C 180,E1 -26460,E2 -26460} C_VEL
LIN {X 0,Y 221.604,Z 617.323,A -85,B 0,C 180,E1 -26464.738,E2 -26464.738} C_VEL
LIN {X 0,Y 223.036,Z 621.129,A -85,B 0,C 180,E1 -26468.95,E2 -26468.95} C_VEL
LIN {X 0,Y 224.607,Z 624.972,A -85,B 0,C 180,E1 -26471.867,E2 -26471.867} C_VEL
LIN {X 0,Y 226.273,Z 628.9,A -85,B 0,C 180,E1 -26474.272,E2 -26474.272} C_VEL
LIN {X 0,Y 228.898,Z 635.728,A -85,B 0,C 180,E1 -26477.415,E2 -26477.415} C_VEL
LIN {X 0,Y 235.447,Z 650.839,A -85,B 0,C 180,E1 -26483.167,E2 -26483.167} C_VEL
LIN {X 0,Y 241.798,Z 660.824,A -85,B 0,C 180,E1 -26487.142,E2 -26487.142} C_VEL
LIN {X 0,Y 249.196,Z 669.88,A -85,B 0,C 180,E1 -26490.823,E2 -26490.823} C_VEL
LIN {X 0,Y 264.387,Z 684.524,A -85,B 0,C 180,E1 -26496.867,E2 -26496.867} C_VEL
LIN {X 0,Y 279.83,Z 696.819,A -85,B 0,C 180,E1 -26501.845,E2 -26501.845} C_VEL
LIN {X 0,Y 288.018,Z 703.08,A -85,B 0,C 180,E1 -26504.55,E2 -26504.55} C_VEL
LIN {X 0,Y 294.971,Z 708.608,A -85,B 0,C 180,E1 -26507.022,E2 -26507.022} C_VEL
LIN {X 0,Y 300.729,Z 713.132,A -85,B 0,C 180,E1 -26509.192,E2 -26509.192} C_VEL
LIN {X 0,Y 307.837,Z 718.471,A -85,B 0,C 180,E1 -26511.991,E2 -26511.991} C_VEL
LIN {X 0,Y 314.096,Z 723.452,A -85,B 0,C 180,E1 -26514.631,E2 -26514.631} C_VEL
LIN {X 0,Y 319.086,Z 726.943,A -85,B 0,C 180,E1 -26516.82,E2 -26516.82} C_VEL
LIN {X 0,Y 324.346,Z 731.417,A -85,B 0,C 180,E1 -26519.364,E2 -26519.364} C_VEL
LIN {X 0,Y 329.792,Z 735.107,A -85,B 0,C 180,E1 -26522.042,E2 -26522.042} C_VEL
LIN {X 0,Y 332.79,Z 737.384,A -85,B 0,C 180,E1 -26523.674,E2 -26523.674} C_VEL
LIN {X 0,Y 337.461,Z 740.952,A -85,B 0,C 180,E1 -26526.397,E2 -26526.397} C_VEL
LIN {X 0,Y 340.495,Z 742.928,A -85,B 0,C 180,E1 -26528.251,E2 -26528.251} C_VEL
LIN {X 0,Y 343.521,Z 744.626,A -85,B 0,C 180,E1 -26530.235,E2 -26530.235} C_VEL
LIN {X 0,Y 346.371,Z 747.192,A -85,B 0,C 180,E1 -26532.485,E2 -26532.485} C_VEL
LIN {X 0,Y 349.244,Z 749.446,A -85,B 0,C 180,E1 -26534.998,E2 -26534.998} C_VEL
LIN {X 0,Y 352.166,Z 751.265,A -85,B 0,C 180,E1 -26537.92,E2 -26537.92} C_VEL
LIN {X 0,Y 354.633,Z 752.305,A -85,B 0,C 180,E1 -26540.878,E2 -26540.878} C_VEL
LIN {X 0,Y 356.089,Z 752.971,A -85,B 0,C 180,E1 -26543.199,E2 -26543.199} C_VEL
LIN {X 0,Y 357.048,Z 753.645,A -85,B 0,C 180,E1 -26545.484,E2 -26545.484} C_VEL
LIN {X 0,Y 357.736,Z 753.733,A -85,B 0,C 180,E1 -26547.748,E2 -26547.748} C_VEL
LIN {X 0,Y 357.874,Z 753.958,A -85,B 0,C 180,E1 -26550,E2 -26550} C_VEL
LIN {X 0,Y 357.706,Z 753.744,A -85,B 0,C 180,E1 -26552.252,E2 -26552.252} C_VEL
LIN {X 0,Y 357.051,Z 753.579,A -85,B 0,C 180,E1 -26554.516,E2 -26554.516} C_VEL
LIN {X 0,Y 356.065,Z 752.998,A -85,B 0,C 180,E1 -26556.801,E2 -26556.801} C_VEL
LIN {X 0,Y 354.598,Z 752.365,A -85,B 0,C 180,E1 -26559.123,E2 -26559.123} C_VEL
LIN {X 0,Y 352.169,Z 751.265,A -85,B 0,C 180,E1 -26562.082,E2 -26562.082} C_VEL
LIN {X 0,Y 349.25,Z 749.389,A -85,B 0,C 180,E1 -26565.006,E2 -26565.006} C_VEL
LIN {X 0,Y 346.107,Z 746.945,A -85,B 0,C 180,E1 -26567.733,E2 -26567.733} C_VEL
LIN {X 0,Y 343.509,Z 744.655,A -85,B 0,C 180,E1 -26569.759,E2 -26569.759} C_VEL
LIN {X 0,Y 340.367,Z 742.878,A -85,B 0,C 180,E1 -26571.818,E2 -26571.818} C_VEL
LIN {X 0,Y 335.237,Z 739.425,A -85,B 0,C 180,E1 -26574.883,E2 -26574.883} C_VEL
LIN {X 0,Y 331.47,Z 736.205,A -85,B 0,C 180,E1 -26577.065,E2 -26577.065} C_VEL
LIN {X 0,Y 326.26,Z 732.777,A -85,B 0,C 180,E1 -26579.698,E2 -26579.698} C_VEL
LIN {X 0,Y 321.038,Z 728.693,A -85,B 0,C 180,E1 -26582.249,E2 -26582.249} C_VEL
LIN {X 0,Y 318.368,Z 726.461,A -85,B 0,C 180,E1 -26583.495,E2 -26583.495} C_VEL
LIN {X 0,Y 312.64,Z 722.376,A -85,B 0,C 180,E1 -26585.977,E2 -26585.977} C_VEL
LIN {X 0,Y 307.03,Z 717.93,A -85,B 0,C 180,E1 -26588.332,E2 -26588.332} C_VEL
LIN {X 0,Y 299.94,Z 712.491,A -85,B 0,C 180,E1 -26591.114,E2 -26591.114} C_VEL
LIN {X 0,Y 293.461,Z 707.396,A -85,B 0,C 180,E1 -26593.533,E2 -26593.533} C_VEL
LIN {X 0,Y 286.439,Z 701.793,A -85,B 0,C 180,E1 -26596,E2 -26596} C_VEL
LIN {X 0,Y 278.624,Z 695.848,A -85,B 0,C 180,E1 -26598.538,E2 -26598.538} C_VEL
LIN {X 0,Y 261.565,Z 682,A -85,B 0,C 180,E1 -26604.164,E2 -26604.164} C_VEL
LIN {X 0,Y 247.142,Z 667.662,A -85,B 0,C 180,E1 -26610.118,E2 -26610.118} C_VEL
LIN {X 0,Y 236.863,Z 653.385,A -85,B 0,C 180,E1 -26615.851,E2 -26615.851} C_VEL
LIN {X 0,Y 230.427,Z 639.95,A -85,B 0,C 180,E1 -26620.992,E2 -26620.992} C_VEL
LIN {X 0,Y 227.825,Z 632.843,A -85,B 0,C 180,E1 -26623.799,E2 -26623.799} C_VEL
LIN {X 0,Y 225.349,Z 626.569,A -85,B 0,C 180,E1 -26627.024,E2 -26627.024} C_VEL
LIN {X 0,Y 223.352,Z 621.955,A -85,B 0,C 180,E1 -26630.378,E2 -26630.378} C_VEL
LIN {X 0,Y 222.497,Z 619.947,A -85,B 0,C 180,E1 -26632.285,E2 -26632.285} C_VEL
LIN {X 0,Y 221.579,Z 617.156,A -85,B 0,C 180,E1 -26635.413,E2 -26635.413} C_VEL
LIN {X 0,Y 221.045,Z 616.251,A -85,B 0,C 180,E1 -26640,E2 -26640} C_VEL
LIN {X 0,Y 221.605,Z 617.308,A -85,B 0,C 180,E1 -26644.32,E2 -26644.32} C_VEL
LIN {X 0,Y 223.071,Z 621.201,A -85,B 0,C 180,E1 -26648.607,E2 -26648.607} C_VEL
LIN {X 0,Y 224.306,Z 624.212,A -85,B 0,C 180,E1 -26650.95,E2 -26650.95} C_VEL
LIN {X 0,Y 226.167,Z 628.575,A -85,B 0,C 180,E1 -26653.706,E2 -26653.706} C_VEL
LIN {X 0,Y 226.709,Z 629.976,A -85,B 0,C 180,E1 -26654.422,E2 -26654.422} C_VEL
LIN {X 0,Y 220.719,Z 684.407,A -85,B 0,C 180,E1 -26655.521,E2 -26655.521} C_VEL
LIN {X 0,Y 217.876,Z 700.176,A -85,B 0,C 180,E1 -26655.923,E2 -26655.923} C_VEL
LIN {X 0,Y 213.079,Z 718.579,A -85,B 0,C 180,E1 -26656.555,E2 -26656.555} C_VEL
LIN {X 0,Y 208.294,Z 732.609,A -85,B 0,C 180,E1 -26657.203,E2 -26657.203} C_VEL
LIN {X 0,Y 203.162,Z 745.244,A -85,B 0,C 180,E1 -26657.96,E2 -26657.96} C_VEL
LIN {X 0,Y 197.138,Z 757.971,A -85,B 0,C 180,E1 -26658.935,E2 -26658.935} C_VEL
LIN {X 0,Y 190.741,Z 769.687,A -85,B 0,C 180,E1 -26660.025,E2 -26660.025} C_VEL
LIN {X 0,Y 183.878,Z 780.811,A -85,B 0,C 180,E1 -26661.312,E2 -26661.312} C_VEL
LIN {X 0,Y 176.358,Z 791.64,A -85,B 0,C 180,E1 -26662.85,E2 -26662.85} C_VEL
LIN {X 0,Y 168.976,Z 801.272,A -85,B 0,C 180,E1 -26664.577,E2 -26664.577} C_VEL
LIN {X 0,Y 161.198,Z 810.519,A -85,B 0,C 180,E1 -26666.652,E2 -26666.652} C_VEL
LIN {X 0,Y 152.815,Z 819.467,A -85,B 0,C 180,E1 -26669.098,E2 -26669.098} C_VEL
LIN {X 0,Y 144.829,Z 827.353,A -85,B 0,C 180,E1 -26671.877,E2 -26671.877} C_VEL
LIN {X 0,Y 137.252,Z 834.317,A -85,B 0,C 180,E1 -26674.989,E2 -26674.989} C_VEL
LIN {X 0,Y 130.112,Z 840.457,A -85,B 0,C 180,E1 -26678.445,E2 -26678.445} C_VEL
LIN {X 0,Y 121.381,Z 847.408,A -85,B 0,C 180,E1 -26683.639,E2 -26683.639} C_VEL
LIN {X 0,Y 113.806,Z 853.173,A -85,B 0,C 180,E1 -26689.579,E2 -26689.579} C_VEL
LIN {X 0,Y 108.978,Z 856.796,A -85,B 0,C 180,E1 -26694.522,E2 -26694.522} C_VEL
LIN {X 0,Y 103.924,Z 860.669,A -85,B 0,C 180,E1 -26701.746,E2 -26701.746} C_VEL
LIN {X 0,Y 100.269,Z 863.54,A -85,B 0,C 180,E1 -26709.485,E2 -26709.485} C_VEL
LIN {X 0,Y 98.323,Z 865.451,A -85,B 0,C 180,E1 -26717.618,E2 -26717.618} C_VEL
LIN {X 0,Y 97.937,Z 866.141,A -85,B 0,C 180,E1 -26721.749,E2 -26721.749} C_VEL
LIN {X 0,Y 98.072,Z 866.638,A -85,B 0,C 180,E1 -26730,E2 -26730} C_VEL
LIN {X 0,Y 97.936,Z 866.141,A -85,B 0,C 180,E1 -26738.252,E2 -26738.252} C_VEL
LIN {X 0,Y 99.041,Z 864.687,A -85,B 0,C 180,E1 -26746.489,E2 -26746.489} C_VEL
LIN {X 0,Y 101.875,Z 862.279,A -85,B 0,C 180,E1 -26754.451,E2 -26754.451} C_VEL
LIN {X 0,Y 107.57,Z 857.841,A -85,B 0,C 180,E1 -26763.733,E2 -26763.733} C_VEL
LIN {X 0,Y 112.106,Z 854.462,A -85,B 0,C 180,E1 -26768.821,E2 -26768.821} C_VEL
LIN {X 0,Y 119.633,Z 848.724,A -85,B 0,C 180,E1 -26775.174,E2 -26775.174} C_VEL
LIN {X 0,Y 125.616,Z 844.09,A -85,B 0,C 180,E1 -26779.05,E2 -26779.05} C_VEL
LIN {X 0,Y 134.867,Z 836.424,A -85,B 0,C 180,E1 -26783.872,E2 -26783.872} C_VEL
LIN {X 0,Y 142.253,Z 829.77,A -85,B 0,C 180,E1 -26787.126,E2 -26787.126} C_VEL
LIN {X 0,Y 150.095,Z 822.222,A -85,B 0,C 180,E1 -26790.022,E2 -26790.022} C_VEL
LIN {X 0,Y 158.308,Z 813.644,A -85,B 0,C 180,E1 -26792.606,E2 -26792.606} C_VEL
LIN {X 0,Y 166.247,Z 804.657,A -85,B 0,C 180,E1 -26794.712,E2 -26794.712} C_VEL
LIN {X 0,Y 174.861,Z 793.65,A -85,B 0,C 180,E1 -26796.834,E2 -26796.834} C_VEL
LIN {X 0,Y 177.586,Z 789.988,A -85,B 0,C 180,E1 -26797.411,E2 -26797.411} C_VEL
LIN {X 0,Y 179.47,Z 787.089,A -85,B 0,C 180,E1 -26798.044,E2 -26798.044} C_VEL
LIN {X 0,Y 181.5,Z 782.614,A -85,B 0,C 180,E1 -26799.526,E2 -26799.526} C_VEL
LIN {X 0,Y 183.464,Z 777.993,A -85,B 0,C 180,E1 -26800.951,E2 -26800.951} C_VEL
LIN {X 0,Y 185.173,Z 774.84,A -85,B 0,C 180,E1 -26801.49,E2 -26801.49} C_VEL
LIN {X 0,Y 192.824,Z 761.768,A -85,B 0,C 180,E1 -26802.72,E2 -26802.72} C_VEL
LIN {X 0,Y 198.693,Z 750.248,A -85,B 0,C 180,E1 -26803.621,E2 -26803.621} C_VEL
LIN {X 0,Y 204.293,Z 737.525,A -85,B 0,C 180,E1 -26804.413,E2 -26804.413} C_VEL
LIN {X 0,Y 209.136,Z 724.537,A -85,B 0,C 180,E1 -26805.043,E2 -26805.043} C_VEL
LIN {X 0,Y 213.194,Z 711.333,A -85,B 0,C 180,E1 -26805.542,E2 -26805.542} C_VEL
LIN {X 0,Y 216.44,Z 697.968,A -85,B 0,C 180,E1 -26805.94,E2 -26805.94} C_VEL
LIN {X 0,Y 218.852,Z 684.416,A -85,B 0,C 180,E1 -26806.28,E2 -26806.28} C_VEL
LIN {X 0,Y 223.262,Z 646.267,A -85,B 0,C 180,E1 -26807.002,E2 -26807.002} C_VEL
LIN {X 0,Y 224.534,Z 634.54,A -85,B 0,C 180,E1 -26807.229,E2 -26807.229} C_VEL
LIN {X 0,Y 222.499,Z 629.38,A -85,B 0,C 180,E1 -26810.684,E2 -26810.684} C_VEL
LIN {X 0,Y 221.505,Z 626.848,A -85,B 0,C 180,E1 -26812.975,E2 -26812.975} C_VEL
LIN {X 0,Y 220.575,Z 624.148,A -85,B 0,C 180,E1 -26816.346,E2 -26816.346} C_VEL
LIN {X 0,Y 220.182,Z 623.282,A -85,B 0,C 180,E1 -26820,E2 -26820} C_VEL
LIN {X 0,Y 220.66,Z 624.278,A -85,B 0,C 180,E1 -26824.442,E2 -26824.442} C_VEL
LIN {X 0,Y 221.925,Z 627.872,A -85,B 0,C 180,E1 -26828.479,E2 -26828.479} C_VEL
LIN {X 0,Y 223.373,Z 631.726,A -85,B 0,C 180,E1 -26831.375,E2 -26831.375} C_VEL
LIN {X 0,Y 224.786,Z 635.263,A -85,B 0,C 180,E1 -26833.561,E2 -26833.561} C_VEL
LIN {X 0,Y 227.095,Z 641.66,A -85,B 0,C 180,E1 -26836.547,E2 -26836.547} C_VEL
LIN {X 0,Y 233.283,Z 656.744,A -85,B 0,C 180,E1 -26842.355,E2 -26842.355} C_VEL
LIN {X 0,Y 239.538,Z 666.931,A -85,B 0,C 180,E1 -26846.466,E2 -26846.466} C_VEL
LIN {X 0,Y 246.595,Z 675.938,A -85,B 0,C 180,E1 -26850.202,E2 -26850.202} C_VEL
LIN {X 0,Y 255.649,Z 685.225,A -85,B 0,C 180,E1 -26854.189,E2 -26854.189} C_VEL
LIN {X 0,Y 266.375,Z 694.869,A -85,B 0,C 180,E1 -26858.245,E2 -26858.245} C_VEL
LIN {X 0,Y 278.779,Z 704.696,A -85,B 0,C 180,E1 -26862.282,E2 -26862.282} C_VEL
LIN {X 0,Y 284.979,Z 709.39,A -85,B 0,C 180,E1 -26864.343,E2 -26864.343} C_VEL
LIN {X 0,Y 292.685,Z 715.489,A -85,B 0,C 180,E1 -26867.085,E2 -26867.085} C_VEL
LIN {X 0,Y 300.163,Z 721.45,A -85,B 0,C 180,E1 -26869.946,E2 -26869.946} C_VEL
LIN {X 0,Y 306.137,Z 725.742,A -85,B 0,C 180,E1 -26872.29,E2 -26872.29} C_VEL
LIN {X 0,Y 311.091,Z 729.79,A -85,B 0,C 180,E1 -26874.418,E2 -26874.418} C_VEL
LIN {X 0,Y 314.997,Z 732.569,A -85,B 0,C 180,E1 -26876.098,E2 -26876.098} C_VEL
LIN {X 0,Y 319.302,Z 736.059,A -85,B 0,C 180,E1 -26878.113,E2 -26878.113} C_VEL
LIN {X 0,Y 324.782,Z 740.119,A -85,B 0,C 180,E1 -26880.779,E2 -26880.779} C_VEL
LIN {X 0,Y 329.972,Z 743.767,A -85,B 0,C 180,E1 -26883.449,E2 -26883.449} C_VEL
LIN {X 0,Y 332.938,Z 746.178,A -85,B 0,C 180,E1 -26885.186,E2 -26885.186} C_VEL
LIN {X 0,Y 337.618,Z 749.325,A -85,B 0,C 180,E1 -26887.995,E2 -26887.995} C_VEL
LIN {X 0,Y 339.862,Z 750.621,A -85,B 0,C 180,E1 -26889.419,E2 -26889.419} C_VEL
LIN {X 0,Y 342.017,Z 752.196,A -85,B 0,C 180,E1 -26890.949,E2 -26890.949} C_VEL
LIN {X 0,Y 345.031,Z 754.756,A -85,B 0,C 180,E1 -26893.431,E2 -26893.431} C_VEL
LIN {X 0,Y 347.809,Z 756.765,A -85,B 0,C 180,E1 -26895.968,E2 -26895.968} C_VEL
LIN {X 0,Y 350.178,Z 758.157,A -85,B 0,C 180,E1 -26898.423,E2 -26898.423} C_VEL
LIN {X 0,Y 352.165,Z 758.936,A -85,B 0,C 180,E1 -26900.814,E2 -26900.814} C_VEL
LIN {X 0,Y 353.752,Z 759.701,A -85,B 0,C 180,E1 -26903.383,E2 -26903.383} C_VEL
LIN {X 0,Y 354.61,Z 760.307,A -85,B 0,C 180,E1 -26905.453,E2 -26905.453} C_VEL
LIN {X 0,Y 355.322,Z 760.405,A -85,B 0,C 180,E1 -26907.733,E2 -26907.733} C_VEL
LIN {X 0,Y 355.456,Z 760.633,A -85,B 0,C 180,E1 -26910,E2 -26910} C_VEL
LIN {X 0,Y 355.292,Z 760.405,A -85,B 0,C 180,E1 -26912.267,E2 -26912.267} C_VEL
LIN {X 0,Y 354.623,Z 760.231,A -85,B 0,C 180,E1 -26914.547,E2 -26914.547} C_VEL
LIN {X 0,Y 353.628,Z 759.639,A -85,B 0,C 180,E1 -26916.848,E2 -26916.848} C_VEL
LIN {X 0,Y 352.137,Z 759.012,A -85,B 0,C 180,E1 -26919.187,E2 -26919.187} C_VEL
LIN {X 0,Y 350.182,Z 758.169,A -85,B 0,C 180,E1 -26921.577,E2 -26921.577} C_VEL
LIN {X 0,Y 347.771,Z 756.73,A -85,B 0,C 180,E1 -26924.068,E2 -26924.068} C_VEL
LIN {X 0,Y 344.854,Z 754.655,A -85,B 0,C 180,E1 -26926.698,E2 -26926.698} C_VEL
LIN {X 0,Y 341.813,Z 752.003,A -85,B 0,C 180,E1 -26929.206,E2 -26929.206} C_VEL
LIN {X 0,Y 339.014,Z 750.191,A -85,B 0,C 180,E1 -26931.113,E2 -26931.113} C_VEL
LIN {X 0,Y 335.129,Z 747.727,A -85,B 0,C 180,E1 -26933.481,E2 -26933.481} C_VEL
LIN {X 0,Y 331.318,Z 744.97,A -85,B 0,C 180,E1 -26935.731,E2 -26935.731} C_VEL
LIN {X 0,Y 328.267,Z 742.382,A -85,B 0,C 180,E1 -26937.456,E2 -26937.456} C_VEL
LIN {X 0,Y 323.163,Z 739.008,A -85,B 0,C 180,E1 -26940.012,E2 -26940.012} C_VEL
LIN {X 0,Y 317.539,Z 734.527,A -85,B 0,C 180,E1 -26942.751,E2 -26942.751} C_VEL
LIN {X 0,Y 311.094,Z 729.777,A -85,B 0,C 180,E1 -26945.583,E2 -26945.583} C_VEL
LIN {X 0,Y 304.582,Z 724.649,A -85,B 0,C 180,E1 -26948.324,E2 -26948.324} C_VEL
LIN {X 0,Y 298.887,Z 720.36,A -85,B 0,C 180,E1 -26950.564,E2 -26950.564} C_VEL
LIN {X 0,Y 292.238,Z 715.124,A -85,B 0,C 180,E1 -26953.074,E2 -26953.074} C_VEL
LIN {X 0,Y 284.56,Z 709.06,A -85,B 0,C 180,E1 -26955.806,E2 -26955.806} C_VEL
LIN {X 0,Y 276.245,Z 702.757,A -85,B 0,C 180,E1 -26958.528,E2 -26958.528} C_VEL
LIN {X 0,Y 256.956,Z 686.582,A -85,B 0,C 180,E1 -26965.272,E2 -26965.272} C_VEL
LIN {X 0,Y 247.022,Z 676.364,A -85,B 0,C 180,E1 -26969.609,E2 -26969.609} C_VEL
LIN {X 0,Y 240.438,Z 668.169,A -85,B 0,C 180,E1 -26973.023,E2 -26973.023} C_VEL
LIN {X 0,Y 234.319,Z 658.645,A -85,B 0,C 180,E1 -26976.884,E2 -26976.884} C_VEL
LIN {X 0,Y 228.632,Z 646.201,A -85,B 0,C 180,E1 -26981.731,E2 -26981.731} C_VEL
LIN {X 0,Y 226.188,Z 639.078,A -85,B 0,C 180,E1 -26984.559,E2 -26984.559} C_VEL
LIN {X 0,Y 223.971,Z 633.069,A -85,B 0,C 180,E1 -26987.672,E2 -26987.672} C_VEL
LIN {X 0,Y 222.19,Z 628.656,A -85,B 0,C 180,E1 -26990.901,E2 -26990.901} C_VEL
LIN {X 0,Y 221.398,Z 626.694,A -85,B 0,C 180,E1 -26992.82,E2 -26992.82} C_VEL
LIN {X 0,Y 220.632,Z 624.156,A -85,B 0,C 180,E1 -26995.712,E2 -26995.712} C_VEL
LIN {X 0,Y 220.179,Z 623.302,A -85,B 0,C 180,E1 -27000,E2 -27000} C_VEL
LIN {X 0,Y 220.687,Z 624.387,A -85,B 0,C 180,E1 -27004.166,E2 -27004.166} C_VEL
LIN {X 0,Y 221.976,Z 628.044,A -85,B 0,C 180,E1 -27008.191,E2 -27008.191} C_VEL
LIN {X 0,Y 223.141,Z 631.103,A -85,B 0,C 180,E1 -27010.549,E2 -27010.549} C_VEL
LIN {X 0,Y 224.532,Z 634.563,A -85,B 0,C 180,E1 -27012.771,E2 -27012.771} C_VEL
LIN {X 0,Y 218.872,Z 684.565,A -85,B 0,C 180,E1 -27013.737,E2 -27013.737} C_VEL
LIN {X 0,Y 215.641,Z 701.965,A -85,B 0,C 180,E1 -27014.172,E2 -27014.172} C_VEL
LIN {X 0,Y 211.166,Z 718.369,A -85,B 0,C 180,E1 -27014.708,E2 -27014.708} C_VEL
LIN {X 0,Y 206.296,Z 732.398,A -85,B 0,C 180,E1 -27015.309,E2 -27015.309} C_VEL
LIN {X 0,Y 201.084,Z 745.026,A -85,B 0,C 180,E1 -27016.03,E2 -27016.03} C_VEL
LIN {X 0,Y 195.169,Z 757.327,A -85,B 0,C 180,E1 -27016.916,E2 -27016.916} C_VEL
LIN {X 0,Y 188.405,Z 769.475,A -85,B 0,C 180,E1 -27017.974,E2 -27017.974} C_VEL
LIN {X 0,Y 181.398,Z 780.6,A -85,B 0,C 180,E1 -27019.204,E2 -27019.204} C_VEL
LIN {X 0,Y 173.7,Z 791.428,A -85,B 0,C 180,E1 -27020.671,E2 -27020.671} C_VEL
LIN {X 0,Y 165.432,Z 801.872,A -85,B 0,C 180,E1 -27022.479,E2 -27022.479} C_VEL
LIN {X 0,Y 158.109,Z 810.307,A -85,B 0,C 180,E1 -27024.327,E2 -27024.327} C_VEL
LIN {X 0,Y 149.45,Z 819.254,A -85,B 0,C 180,E1 -27026.688,E2 -27026.688} C_VEL
LIN {X 0,Y 141.154,Z 827.14,A -85,B 0,C 180,E1 -27029.391,E2 -27029.391} C_VEL
LIN {X 0,Y 133.226,Z 834.103,A -85,B 0,C 180,E1 -27032.433,E2 -27032.433} C_VEL
LIN {X 0,Y 125.761,Z 840.244,A -85,B 0,C 180,E1 -27035.875,E2 -27035.875} C_VEL
LIN {X 0,Y 116.515,Z 847.193,A -85,B 0,C 180,E1 -27041.065,E2 -27041.065} C_VEL
LIN {X 0,Y 108.402,Z 852.959,A -85,B 0,C 180,E1 -27047.099,E2 -27047.099} C_VEL
LIN {X 0,Y 103.182,Z 856.583,A -85,B 0,C 180,E1 -27052.193,E2 -27052.193} C_VEL
LIN {X 0,Y 97.553,Z 860.493,A -85,B 0,C 180,E1 -27059.829,E2 -27059.829} C_VEL
LIN {X 0,Y 93.576,Z 863.328,A -85,B 0,C 180,E1 -27067.944,E2 -27067.944} C_VEL
LIN {X 0,Y 91.324,Z 865.239,A -85,B 0,C 180,E1 -27076.652,E2 -27076.652} C_VEL
LIN {X 0,Y 90.884,Z 865.93,A -85,B 0,C 180,E1 -27081.103,E2 -27081.103} C_VEL
LIN {X 0,Y 90.97,Z 866.428,A -85,B 0,C 180,E1 -27090,E2 -27090} C_VEL
LIN {X 0,Y 90.861,Z 865.93,A -85,B 0,C 180,E1 -27098.899,E2 -27098.899} C_VEL
LIN {X 0,Y 92.179,Z 864.475,A -85,B 0,C 180,E1 -27107.756,E2 -27107.756} C_VEL
LIN {X 0,Y 95.381,Z 862.067,A -85,B 0,C 180,E1 -27116.237,E2 -27116.237} C_VEL
LIN {X 0,Y 101.651,Z 857.628,A -85,B 0,C 180,E1 -27125.991,E2 -27125.991} C_VEL
LIN {X 0,Y 106.58,Z 854.249,A -85,B 0,C 180,E1 -27131.254,E2 -27131.254} C_VEL
LIN {X 0,Y 114.349,Z 848.738,A -85,B 0,C 180,E1 -27137.52,E2 -27137.52} C_VEL
LIN {X 0,Y 121.019,Z 843.877,A -85,B 0,C 180,E1 -27141.626,E2 -27141.626} C_VEL
LIN {X 0,Y 130.735,Z 836.211,A -85,B 0,C 180,E1 -27146.431,E2 -27146.431} C_VEL
LIN {X 0,Y 138.471,Z 829.557,A -85,B 0,C 180,E1 -27149.632,E2 -27149.632} C_VEL
LIN {X 0,Y 146.628,Z 822.009,A -85,B 0,C 180,E1 -27152.461,E2 -27152.461} C_VEL
LIN {X 0,Y 155.15,Z 813.433,A -85,B 0,C 180,E1 -27154.95,E2 -27154.95} C_VEL
LIN {X 0,Y 163.001,Z 804.813,A -85,B 0,C 180,E1 -27156.917,E2 -27156.917} C_VEL
LIN {X 0,Y 172.175,Z 793.439,A -85,B 0,C 180,E1 -27159.021,E2 -27159.021} C_VEL
LIN {X 0,Y 179.835,Z 782.883,A -85,B 0,C 180,E1 -27160.526,E2 -27160.526} C_VEL
LIN {X 0,Y 185.173,Z 774.84,A -85,B 0,C 180,E1 -27161.49,E2 -27161.49} C_VEL
LIN {X 0,Y 187.85,Z 770.065,A -85,B 0,C 180,E1 -27162.155,E2 -27162.155} C_VEL
LIN {X 0,Y 194.877,Z 754.406,A -85,B 0,C 180,E1 -27165.122,E2 -27165.122} C_VEL
LIN {X 0,Y 197.176,Z 749.24,A -85,B 0,C 180,E1 -27165.659,E2 -27165.659} C_VEL
LIN {X 0,Y 202.904,Z 736.29,A -85,B 0,C 180,E1 -27166.404,E2 -27166.404} C_VEL
LIN {X 0,Y 207.828,Z 723.094,A -85,B 0,C 180,E1 -27166.986,E2 -27166.986} C_VEL
LIN {X 0,Y 211.742,Z 710.358,A -85,B 0,C 180,E1 -27167.424,E2 -27167.424} C_VEL
LIN {X 0,Y 214.825,Z 697.758,A -85,B 0,C 180,E1 -27167.778,E2 -27167.778} C_VEL
LIN {X 0,Y 217.276,Z 684.206,A -85,B 0,C 180,E1 -27168.1,E2 -27168.1} C_VEL
LIN {X 0,Y 221.888,Z 645.081,A -85,B 0,C 180,E1 -27168.799,E2 -27168.799} C_VEL
LIN {X 0,Y 222.495,Z 639.211,A -85,B 0,C 180,E1 -27168.964,E2 -27168.964} C_VEL
LIN {X 0,Y 220.998,Z 635.182,A -85,B 0,C 180,E1 -27171.973,E2 -27171.973} C_VEL
LIN {X 0,Y 220.343,Z 633.415,A -85,B 0,C 180,E1 -27173.73,E2 -27173.73} C_VEL
LIN {X 0,Y 219.71,Z 631.206,A -85,B 0,C 180,E1 -27176.332,E2 -27176.332} C_VEL
LIN {X 0,Y 219.316,Z 630.33,A -85,B 0,C 180,E1 -27180,E2 -27180} C_VEL
LIN {X 0,Y 219.745,Z 631.395,A -85,B 0,C 180,E1 -27184.302,E2 -27184.302} C_VEL
LIN {X 0,Y 220.819,Z 634.677,A -85,B 0,C 180,E1 -27187.997,E2 -27187.997} C_VEL
LIN {X 0,Y 222.131,Z 638.378,A -85,B 0,C 180,E1 -27190.827,E2 -27190.827} C_VEL
LIN {X 0,Y 223.374,Z 641.696,A -85,B 0,C 180,E1 -27192.896,E2 -27192.896} C_VEL
LIN {X 0,Y 225.486,Z 648.064,A -85,B 0,C 180,E1 -27195.847,E2 -27195.847} C_VEL
LIN {X 0,Y 231.283,Z 662.86,A -85,B 0,C 180,E1 -27201.619,E2 -27201.619} C_VEL
LIN {X 0,Y 236.972,Z 672.589,A -85,B 0,C 180,E1 -27205.587,E2 -27205.587} C_VEL
LIN {X 0,Y 244.401,Z 682.431,A -85,B 0,C 180,E1 -27209.765,E2 -27209.765} C_VEL
LIN {X 0,Y 257.683,Z 696.255,A -85,B 0,C 180,E1 -27215.812,E2 -27215.812} C_VEL
LIN {X 0,Y 274.404,Z 710.106,A -85,B 0,C 180,E1 -27221.751,E2 -27221.751} C_VEL
LIN {X 0,Y 281.966,Z 715.867,A -85,B 0,C 180,E1 -27224.258,E2 -27224.258} C_VEL
LIN {X 0,Y 289.138,Z 721.534,A -85,B 0,C 180,E1 -27226.819,E2 -27226.819} C_VEL
LIN {X 0,Y 296.081,Z 726.987,A -85,B 0,C 180,E1 -27229.426,E2 -27229.426} C_VEL
LIN {X 0,Y 302.85,Z 731.96,A -85,B 0,C 180,E1 -27232.092,E2 -27232.092} C_VEL
LIN {X 0,Y 309.389,Z 737.159,A -85,B 0,C 180,E1 -27234.861,E2 -27234.861} C_VEL
LIN {X 0,Y 313.919,Z 740.386,A -85,B 0,C 180,E1 -27236.84,E2 -27236.84} C_VEL
LIN {X 0,Y 319.663,Z 745.025,A -85,B 0,C 180,E1 -27239.625,E2 -27239.625} C_VEL
LIN {X 0,Y 323.33,Z 747.544,A -85,B 0,C 180,E1 -27241.433,E2 -27241.433} C_VEL
LIN {X 0,Y 326.627,Z 749.888,A -85,B 0,C 180,E1 -27243.138,E2 -27243.138} C_VEL
LIN {X 0,Y 331.236,Z 753.493,A -85,B 0,C 180,E1 -27245.831,E2 -27245.831} C_VEL
LIN {X 0,Y 334.512,Z 755.646,A -85,B 0,C 180,E1 -27247.78,E2 -27247.78} C_VEL
LIN {X 0,Y 337.407,Z 757.363,A -85,B 0,C 180,E1 -27249.605,E2 -27249.605} C_VEL
LIN {X 0,Y 340.484,Z 759.895,A -85,B 0,C 180,E1 -27251.964,E2 -27251.964} C_VEL
LIN {X 0,Y 343.538,Z 762.258,A -85,B 0,C 180,E1 -27254.577,E2 -27254.577} C_VEL
LIN {X 0,Y 346.14,Z 764.029,A -85,B 0,C 180,E1 -27257.095,E2 -27257.095} C_VEL
LIN {X 0,Y 348.436,Z 765.075,A -85,B 0,C 180,E1 -27259.541,E2 -27259.541} C_VEL
LIN {X 0,Y 350.176,Z 765.884,A -85,B 0,C 180,E1 -27261.924,E2 -27261.924} C_VEL
LIN {X 0,Y 351.431,Z 766.534,A -85,B 0,C 180,E1 -27264.261,E2 -27264.261} C_VEL
LIN {X 0,Y 352.281,Z 766.944,A -85,B 0,C 180,E1 -27266.569,E2 -27266.569} C_VEL
LIN {X 0,Y 352.74,Z 767.07,A -85,B 0,C 180,E1 -27268.858,E2 -27268.858} C_VEL
LIN {X 0,Y 352.713,Z 767.078,A -85,B 0,C 180,E1 -27271.142,E2 -27271.142} C_VEL
LIN {X 0,Y 352.16,Z 766.935,A -85,B 0,C 180,E1 -27273.776,E2 -27273.776} C_VEL
LIN {X 0,Y 351.427,Z 766.536,A -85,B 0,C 180,E1 -27275.739,E2 -27275.739} C_VEL
LIN {X 0,Y 350.192,Z 765.875,A -85,B 0,C 180,E1 -27278.076,E2 -27278.076} C_VEL
LIN {X 0,Y 348.42,Z 765.152,A -85,B 0,C 180,E1 -27280.459,E2 -27280.459} C_VEL
LIN {X 0,Y 346.138,Z 763.947,A -85,B 0,C 180,E1 -27282.946,E2 -27282.946} C_VEL
LIN {X 0,Y 343.174,Z 761.995,A -85,B 0,C 180,E1 -27285.736,E2 -27285.736} C_VEL
LIN {X 0,Y 340.295,Z 759.686,A -85,B 0,C 180,E1 -27288.193,E2 -27288.193} C_VEL
LIN {X 0,Y 337.397,Z 757.373,A -85,B 0,C 180,E1 -27290.39,E2 -27290.39} C_VEL
LIN {X 0,Y 334.309,Z 755.547,A -85,B 0,C 180,E1 -27292.335,E2 -27292.335} C_VEL
LIN {X 0,Y 329.433,Z 752.206,A -85,B 0,C 180,E1 -27295.256,E2 -27295.256} C_VEL
LIN {X 0,Y 325.222,Z 748.718,A -85,B 0,C 180,E1 -27297.626,E2 -27297.626} C_VEL
LIN {X 0,Y 319.663,Z 745.013,A -85,B 0,C 180,E1 -27300.375,E2 -27300.375} C_VEL
LIN {X 0,Y 313.867,Z 740.411,A -85,B 0,C 180,E1 -27303.168,E2 -27303.168} C_VEL
LIN {X 0,Y 307.866,Z 735.994,A -85,B 0,C 180,E1 -27305.788,E2 -27305.788} C_VEL
LIN {X 0,Y 301.017,Z 730.633,A -85,B 0,C 180,E1 -27308.653,E2 -27308.653} C_VEL
LIN {X 0,Y 294.267,Z 725.488,A -85,B 0,C 180,E1 -27311.275,E2 -27311.275} C_VEL
LIN {X 0,Y 287.385,Z 720.172,A -85,B 0,C 180,E1 -27313.829,E2 -27313.829} C_VEL
LIN {X 0,Y 280.131,Z 714.362,A -85,B 0,C 180,E1 -27316.376,E2 -27316.376} C_VEL
LIN {X 0,Y 271.148,Z 707.517,A -85,B 0,C 180,E1 -27319.306,E2 -27319.306} C_VEL
LIN {X 0,Y 254.445,Z 693.128,A -85,B 0,C 180,E1 -27325.54,E2 -27325.54} C_VEL
LIN {X 0,Y 242.465,Z 680.187,A -85,B 0,C 180,E1 -27331.237,E2 -27331.237} C_VEL
LIN {X 0,Y 232.764,Z 665.739,A -85,B 0,C 180,E1 -27337.242,E2 -27337.242} C_VEL
LIN {X 0,Y 226.687,Z 651.855,A -85,B 0,C 180,E1 -27342.697,E2 -27342.697} C_VEL
LIN {X 0,Y 224.474,Z 644.937,A -85,B 0,C 180,E1 -27345.495,E2 -27345.495} C_VEL
LIN {X 0,Y 222.588,Z 639.467,A -85,B 0,C 180,E1 -27348.388,E2 -27348.388} C_VEL
LIN {X 0,Y 220.86,Z 634.806,A -85,B 0,C 180,E1 -27351.895,E2 -27351.895} C_VEL
LIN {X 0,Y 219.692,Z 631.148,A -85,B 0,C 180,E1 -27356.013,E2 -27356.013} C_VEL
LIN {X 0,Y 219.313,Z 630.354,A -85,B 0,C 180,E1 -27360,E2 -27360} C_VEL
LIN {X 0,Y 219.751,Z 631.372,A -85,B 0,C 180,E1 -27363.897,E2 -27363.897} C_VEL
LIN {X 0,Y 220.893,Z 634.892,A -85,B 0,C 180,E1 -27367.772,E2 -27367.772} C_VEL
LIN {X 0,Y 221.979,Z 637.939,A -85,B 0,C 180,E1 -27370.123,E2 -27370.123} C_VEL
LIN {X 0,Y 222.516,Z 639.372,A -85,B 0,C 180,E1 -27371.09,E2 -27371.09} C_VEL
LIN {X 0,Y 217.294,Z 684.382,A -85,B 0,C 180,E1 -27371.92,E2 -27371.92} C_VEL
LIN {X 0,Y 214.009,Z 701.755,A -85,B 0,C 180,E1 -27372.324,E2 -27372.324} C_VEL
LIN {X 0,Y 209.469,Z 718.159,A -85,B 0,C 180,E1 -27372.821,E2 -27372.821} C_VEL
LIN {X 0,Y 204.531,Z 732.188,A -85,B 0,C 180,E1 -27373.384,E2 -27373.384} C_VEL
LIN {X 0,Y 199.233,Z 744.816,A -85,B 0,C 180,E1 -27374.058,E2 -27374.058} C_VEL
LIN {X 0,Y 193.836,Z 755.954,A -85,B 0,C 180,E1 -27374.8,E2 -27374.8} C_VEL
LIN {X 0,Y 187.137,Z 767.961,A -85,B 0,C 180,E1 -27375.776,E2 -27375.776} C_VEL
LIN {X 0,Y 179.959,Z 779.245,A -85,B 0,C 180,E1 -27376.906,E2 -27376.906} C_VEL
LIN {X 0,Y 172.088,Z 790.211,A -85,B 0,C 180,E1 -27378.287,E2 -27378.287} C_VEL
LIN {X 0,Y 164.352,Z 799.893,A -85,B 0,C 180,E1 -27379.824,E2 -27379.824} C_VEL
LIN {X 0,Y 155.287,Z 810.095,A -85,B 0,C 180,E1 -27381.911,E2 -27381.911} C_VEL
LIN {X 0,Y 146.369,Z 819.042,A -85,B 0,C 180,E1 -27384.178,E2 -27384.178} C_VEL
LIN {X 0,Y 137.754,Z 826.927,A -85,B 0,C 180,E1 -27386.773,E2 -27386.773} C_VEL
LIN {X 0,Y 129.489,Z 833.889,A -85,B 0,C 180,E1 -27389.73,E2 -27389.73} C_VEL
LIN {X 0,Y 121.673,Z 840.031,A -85,B 0,C 180,E1 -27393.121,E2 -27393.121} C_VEL
LIN {X 0,Y 111.91,Z 846.98,A -85,B 0,C 180,E1 -27398.28,E2 -27398.28} C_VEL
LIN {X 0,Y 105.28,Z 851.456,A -85,B 0,C 180,E1 -27402.752,E2 -27402.752} C_VEL
LIN {X 0,Y 97.568,Z 856.369,A -85,B 0,C 180,E1 -27409.589,E2 -27409.589} C_VEL
LIN {X 0,Y 90.973,Z 860.527,A -85,B 0,C 180,E1 -27418.19,E2 -27418.19} C_VEL
LIN {X 0,Y 86.967,Z 863.115,A -85,B 0,C 180,E1 -27426.168,E2 -27426.168} C_VEL
LIN {X 0,Y 84.36,Z 865.027,A -85,B 0,C 180,E1 -27435.527,E2 -27435.527} C_VEL
LIN {X 0,Y 83.829,Z 865.719,A -85,B 0,C 180,E1 -27440.348,E2 -27440.348} C_VEL
LIN {X 0,Y 83.875,Z 866.219,A -85,B 0,C 180,E1 -27450,E2 -27450} C_VEL
LIN {X 0,Y 83.811,Z 865.719,A -85,B 0,C 180,E1 -27459.654,E2 -27459.654} C_VEL
LIN {X 0,Y 85.369,Z 864.263,A -85,B 0,C 180,E1 -27469.226,E2 -27469.226} C_VEL
LIN {X 0,Y 88.992,Z 861.854,A -85,B 0,C 180,E1 -27478.283,E2 -27478.283} C_VEL
LIN {X 0,Y 95.885,Z 857.414,A -85,B 0,C 180,E1 -27488.536,E2 -27488.536} C_VEL
LIN {X 0,Y 101.27,Z 854.035,A -85,B 0,C 180,E1 -27493.945,E2 -27493.945} C_VEL
LIN {X 0,Y 109.612,Z 848.525,A -85,B 0,C 180,E1 -27500.299,E2 -27500.299} C_VEL
LIN {X 0,Y 116.668,Z 843.664,A -85,B 0,C 180,E1 -27504.411,E2 -27504.411} C_VEL
LIN {X 0,Y 126.876,Z 835.997,A -85,B 0,C 180,E1 -27509.156,E2 -27509.156} C_VEL
LIN {X 0,Y 134.972,Z 829.344,A -85,B 0,C 180,E1 -27512.273,E2 -27512.273} C_VEL
LIN {X 0,Y 143.434,Z 821.795,A -85,B 0,C 180,E1 -27515.018,E2 -27515.018} C_VEL
LIN {X 0,Y 152.264,Z 813.222,A -85,B 0,C 180,E1 -27517.385,E2 -27517.385} C_VEL
LIN {X 0,Y 161.025,Z 803.759,A -85,B 0,C 180,E1 -27519.455,E2 -27519.455} C_VEL
LIN {X 0,Y 169.737,Z 793.227,A -85,B 0,C 180,E1 -27521.285,E2 -27521.285} C_VEL
LIN {X 0,Y 177.579,Z 782.672,A -85,B 0,C 180,E1 -27522.701,E2 -27522.701} C_VEL
LIN {X 0,Y 184.73,Z 771.872,A -85,B 0,C 180,E1 -27523.864,E2 -27523.864} C_VEL
LIN {X 0,Y 191.271,Z 760.714,A -85,B 0,C 180,E1 -27524.84,E2 -27524.84} C_VEL
LIN {X 0,Y 197.176,Z 749.24,A -85,B 0,C 180,E1 -27525.659,E2 -27525.659} C_VEL
LIN {X 0,Y 199.484,Z 744.042,A -85,B 0,C 180,E1 -27526.138,E2 -27526.138} C_VEL
LIN {X 0,Y 205.108,Z 727.044,A -85,B 0,C 180,E1 -27528.538,E2 -27528.538} C_VEL
LIN {X 0,Y 206.782,Z 721.6,A -85,B 0,C 180,E1 -27528.948,E2 -27528.948} C_VEL
LIN {X 0,Y 210.518,Z 709.382,A -85,B 0,C 180,E1 -27529.335,E2 -27529.335} C_VEL
LIN {X 0,Y 213.643,Z 696.549,A -85,B 0,C 180,E1 -27529.664,E2 -27529.664} C_VEL
LIN {X 0,Y 216.029,Z 683.278,A -85,B 0,C 180,E1 -27529.956,E2 -27529.956} C_VEL
LIN {X 0,Y 220.669,Z 644.232,A -85,B 0,C 180,E1 -27530.654,E2 -27530.654} C_VEL
LIN {X 0,Y 219.521,Z 640.709,A -85,B 0,C 180,E1 -27533.551,E2 -27533.551} C_VEL
LIN {X 0,Y 218.747,Z 638.146,A -85,B 0,C 180,E1 -27536.776,E2 -27536.776} C_VEL
LIN {X 0,Y 218.451,Z 637.38,A -85,B 0,C 180,E1 -27540,E2 -27540} C_VEL
LIN {X 0,Y 218.81,Z 638.35,A -85,B 0,C 180,E1 -27544.001,E2 -27544.001} C_VEL
LIN {X 0,Y 219.743,Z 641.464,A -85,B 0,C 180,E1 -27547.537,E2 -27547.537} C_VEL
LIN {X 0,Y 221.348,Z 646.142,A -85,B 0,C 180,E1 -27551.081,E2 -27551.081} C_VEL
LIN {X 0,Y 223.198,Z 652.057,A -85,B 0,C 180,E1 -27554.124,E2 -27554.124} C_VEL
LIN {X 0,Y 229.573,Z 669.496,A -85,B 0,C 180,E1 -27561.082,E2 -27561.082} C_VEL
LIN {X 0,Y 234.79,Z 678.908,A -85,B 0,C 180,E1 -27565.006,E2 -27565.006} C_VEL
LIN {X 0,Y 241.195,Z 687.971,A -85,B 0,C 180,E1 -27568.933,E2 -27568.933} C_VEL
LIN {X 0,Y 253.709,Z 701.621,A -85,B 0,C 180,E1 -27575.085,E2 -27575.085} C_VEL
LIN {X 0,Y 270.565,Z 715.968,A -85,B 0,C 180,E1 -27581.48,E2 -27581.48} C_VEL
LIN {X 0,Y 278.177,Z 721.768,A -85,B 0,C 180,E1 -27584.008,E2 -27584.008} C_VEL
LIN {X 0,Y 285.247,Z 727.354,A -85,B 0,C 180,E1 -27586.518,E2 -27586.518} C_VEL
LIN {X 0,Y 292.424,Z 732.969,A -85,B 0,C 180,E1 -27589.206,E2 -27589.206} C_VEL
LIN {X 0,Y 298.986,Z 737.81,A -85,B 0,C 180,E1 -27591.768,E2 -27591.768} C_VEL
LIN {X 0,Y 304.193,Z 741.998,A -85,B 0,C 180,E1 -27593.961,E2 -27593.961} C_VEL
LIN {X 0,Y 310.735,Z 746.733,A -85,B 0,C 180,E1 -27596.807,E2 -27596.807} C_VEL
LIN {X 0,Y 315.711,Z 750.785,A -85,B 0,C 180,E1 -27599.204,E2 -27599.204} C_VEL
LIN {X 0,Y 320.188,Z 753.902,A -85,B 0,C 180,E1 -27601.399,E2 -27601.399} C_VEL
LIN {X 0,Y 323.323,Z 756.108,A -85,B 0,C 180,E1 -27603.024,E2 -27603.024} C_VEL
LIN {X 0,Y 326.361,Z 758.584,A -85,B 0,C 180,E1 -27604.747,E2 -27604.747} C_VEL
LIN {X 0,Y 331.068,Z 761.786,A -85,B 0,C 180,E1 -27607.536,E2 -27607.536} C_VEL
LIN {X 0,Y 333.466,Z 763.204,A -85,B 0,C 180,E1 -27609.006,E2 -27609.006} C_VEL
LIN {X 0,Y 335.552,Z 764.655,A -85,B 0,C 180,E1 -27610.475,E2 -27610.475} C_VEL
LIN {X 0,Y 338.819,Z 767.381,A -85,B 0,C 180,E1 -27613.119,E2 -27613.119} C_VEL
LIN {X 0,Y 341.705,Z 769.503,A -85,B 0,C 180,E1 -27615.712,E2 -27615.712} C_VEL
LIN {X 0,Y 344.373,Z 771.071,A -85,B 0,C 180,E1 -27618.401,E2 -27618.401} C_VEL
LIN {X 0,Y 346.26,Z 771.845,A -85,B 0,C 180,E1 -27620.655,E2 -27620.655} C_VEL
LIN {X 0,Y 347.805,Z 772.545,A -85,B 0,C 180,E1 -27623.036,E2 -27623.036} C_VEL
LIN {X 0,Y 348.809,Z 773.224,A -85,B 0,C 180,E1 -27625.377,E2 -27625.377} C_VEL
LIN {X 0,Y 349.556,Z 773.37,A -85,B 0,C 180,E1 -27627.696,E2 -27627.696} C_VEL
LIN {X 0,Y 349.697,Z 773.588,A -85,B 0,C 180,E1 -27630,E2 -27630} C_VEL
LIN {X 0,Y 349.523,Z 773.374,A -85,B 0,C 180,E1 -27632.305,E2 -27632.305} C_VEL
LIN {X 0,Y 348.831,Z 773.162,A -85,B 0,C 180,E1 -27634.622,E2 -27634.622} C_VEL
LIN {X 0,Y 347.418,Z 772.411,A -85,B 0,C 180,E1 -27637.598,E2 -27637.598} C_VEL
LIN {X 0,Y 346.255,Z 771.909,A -85,B 0,C 180,E1 -27639.345,E2 -27639.345} C_VEL
LIN {X 0,Y 344.222,Z 770.988,A -85,B 0,C 180,E1 -27641.781,E2 -27641.781} C_VEL
LIN {X 0,Y 341.356,Z 769.266,A -85,B 0,C 180,E1 -27644.614,E2 -27644.614} C_VEL
LIN {X 0,Y 338.413,Z 767.121,A -85,B 0,C 180,E1 -27647.197,E2 -27647.197} C_VEL
LIN {X 0,Y 335.469,Z 764.581,A -85,B 0,C 180,E1 -27649.584,E2 -27649.584} C_VEL
LIN {X 0,Y 332.518,Z 762.686,A -85,B 0,C 180,E1 -27651.571,E2 -27651.571} C_VEL
LIN {X 0,Y 328.495,Z 760.133,A -85,B 0,C 180,E1 -27653.984,E2 -27653.984} C_VEL
LIN {X 0,Y 324.631,Z 757.216,A -85,B 0,C 180,E1 -27656.242,E2 -27656.242} C_VEL
LIN {X 0,Y 319.521,Z 753.408,A -85,B 0,C 180,E1 -27658.94,E2 -27658.94} C_VEL
LIN {X 0,Y 315.699,Z 750.782,A -85,B 0,C 180,E1 -27660.798,E2 -27660.798} C_VEL
LIN {X 0,Y 309.216,Z 745.624,A -85,B 0,C 180,E1 -27663.88,E2 -27663.88} C_VEL
LIN {X 0,Y 302.604,Z 740.772,A -85,B 0,C 180,E1 -27666.711,E2 -27666.711} C_VEL
LIN {X 0,Y 297.569,Z 736.771,A -85,B 0,C 180,E1 -27668.796,E2 -27668.796} C_VEL
LIN {X 0,Y 290.72,Z 731.569,A -85,B 0,C 180,E1 -27671.462,E2 -27671.462} C_VEL
LIN {X 0,Y 284.467,Z 726.713,A -85,B 0,C 180,E1 -27673.769,E2 -27673.769} C_VEL
LIN {X 0,Y 278.181,Z 721.732,A -85,B 0,C 180,E1 -27675.992,E2 -27675.992} C_VEL
LIN {X 0,Y 270.569,Z 715.955,A -85,B 0,C 180,E1 -27678.521,E2 -27678.521} C_VEL
LIN {X 0,Y 252.402,Z 700.327,A -85,B 0,C 180,E1 -27685.497,E2 -27685.497} C_VEL
LIN {X 0,Y 240.566,Z 687.198,A -85,B 0,C 180,E1 -27691.42,E2 -27691.42} C_VEL
LIN {X 0,Y 232.304,Z 674.846,A -85,B 0,C 180,E1 -27696.756,E2 -27696.756} C_VEL
LIN {X 0,Y 226.168,Z 661.481,A -85,B 0,C 180,E1 -27702.116,E2 -27702.116} C_VEL
LIN {X 0,Y 222.937,Z 651.19,A -85,B 0,C 180,E1 -27706.266,E2 -27706.266} C_VEL
LIN {X 0,Y 221.29,Z 646.032,A -85,B 0,C 180,E1 -27709.015,E2 -27709.015} C_VEL
LIN {X 0,Y 219.865,Z 641.911,A -85,B 0,C 180,E1 -27712.112,E2 -27712.112} C_VEL
LIN {X 0,Y 219.112,Z 639.65,A -85,B 0,C 180,E1 -27714.479,E2 -27714.479} C_VEL
LIN {X 0,Y 218.759,Z 638.131,A -85,B 0,C 180,E1 -27716.316,E2 -27716.316} C_VEL
LIN {X 0,Y 218.447,Z 637.407,A -85,B 0,C 180,E1 -27720,E2 -27720} C_VEL
LIN {X 0,Y 218.826,Z 638.419,A -85,B 0,C 180,E1 -27723.683,E2 -27723.683} C_VEL
LIN {X 0,Y 219.825,Z 641.723,A -85,B 0,C 180,E1 -27727.348,E2 -27727.348} C_VEL
LIN {X 0,Y 220.67,Z 644.306,A -85,B 0,C 180,E1 -27729.363,E2 -27729.363} C_VEL
LIN {X 0,Y 215.913,Z 684.355,A -85,B 0,C 180,E1 -27730.079,E2 -27730.079} C_VEL
LIN {X 0,Y 212.401,Z 702.461,A -85,B 0,C 180,E1 -27730.479,E2 -27730.479} C_VEL
LIN {X 0,Y 207.59,Z 719.182,A -85,B 0,C 180,E1 -27730.955,E2 -27730.955} C_VEL
LIN {X 0,Y 203.006,Z 731.978,A -85,B 0,C 180,E1 -27731.436,E2 -27731.436} C_VEL
LIN {X 0,Y 197.623,Z 744.605,A -85,B 0,C 180,E1 -27732.055,E2 -27732.055} C_VEL
LIN {X 0,Y 191.548,Z 756.824,A -85,B 0,C 180,E1 -27732.822,E2 -27732.822} C_VEL
LIN {X 0,Y 184.508,Z 769.054,A -85,B 0,C 180,E1 -27733.765,E2 -27733.765} C_VEL
LIN {X 0,Y 177.202,Z 780.176,A -85,B 0,C 180,E1 -27734.825,E2 -27734.825} C_VEL
LIN {X 0,Y 169.177,Z 791.005,A -85,B 0,C 180,E1 -27736.128,E2 -27736.128} C_VEL
LIN {X 0,Y 160.644,Z 801.286,A -85,B 0,C 180,E1 -27737.719,E2 -27737.719} C_VEL
LIN {X 0,Y 152.746,Z 809.882,A -85,B 0,C 180,E1 -27739.403,E2 -27739.403} C_VEL
LIN {X 0,Y 143.563,Z 818.829,A -85,B 0,C 180,E1 -27741.549,E2 -27741.549} C_VEL
LIN {X 0,Y 134.657,Z 826.713,A -85,B 0,C 180,E1 -27744.03,E2 -27744.03} C_VEL
LIN {X 0,Y 126.068,Z 833.676,A -85,B 0,C 180,E1 -27746.881,E2 -27746.881} C_VEL
LIN {X 0,Y 117.896,Z 839.818,A -85,B 0,C 180,E1 -27750.192,E2 -27750.192} C_VEL
LIN {X 0,Y 107.591,Z 846.766,A -85,B 0,C 180,E1 -27755.264,E2 -27755.264} C_VEL
LIN {X 0,Y 98.312,Z 852.532,A -85,B 0,C 180,E1 -27761.358,E2 -27761.358} C_VEL
LIN {X 0,Y 92.178,Z 856.155,A -85,B 0,C 180,E1 -27766.672,E2 -27766.672} C_VEL
LIN {X 0,Y 84.566,Z 860.525,A -85,B 0,C 180,E1 -27776.21,E2 -27776.21} C_VEL
LIN {X 0,Y 80.445,Z 862.903,A -85,B 0,C 180,E1 -27784.099,E2 -27784.099} C_VEL
LIN {X 0,Y 77.445,Z 864.815,A -85,B 0,C 180,E1 -27794.202,E2 -27794.202} C_VEL
LIN {X 0,Y 76.803,Z 865.508,A -85,B 0,C 180,E1 -27799.455,E2 -27799.455} C_VEL
LIN {X 0,Y 76.771,Z 866.009,A -85,B 0,C 180,E1 -27810,E2 -27810} C_VEL
LIN {X 0,Y 76.76,Z 865.507,A -85,B 0,C 180,E1 -27820.551,E2 -27820.551} C_VEL
LIN {X 0,Y 78.628,Z 864.05,A -85,B 0,C 180,E1 -27830.948,E2 -27830.948} C_VEL
LIN {X 0,Y 82.714,Z 861.641,A -85,B 0,C 180,E1 -27840.65,E2 -27840.65} C_VEL
LIN {X 0,Y 90.349,Z 857.2,A -85,B 0,C 180,E1 -27851.389,E2 -27851.389} C_VEL
LIN {X 0,Y 96.191,Z 853.822,A -85,B 0,C 180,E1 -27856.938,E2 -27856.938} C_VEL
LIN {X 0,Y 105.156,Z 848.312,A -85,B 0,C 180,E1 -27863.32,E2 -27863.32} C_VEL
LIN {X 0,Y 112.625,Z 843.451,A -85,B 0,C 180,E1 -27867.394,E2 -27867.394} C_VEL
LIN {X 0,Y 123.329,Z 835.784,A -85,B 0,C 180,E1 -27872.038,E2 -27872.038} C_VEL
LIN {X 0,Y 131.773,Z 829.131,A -85,B 0,C 180,E1 -27875.048,E2 -27875.048} C_VEL
LIN {X 0,Y 140.552,Z 821.583,A -85,B 0,C 180,E1 -27877.673,E2 -27877.673} C_VEL
LIN {X 0,Y 149.661,Z 813.01,A -85,B 0,C 180,E1 -27879.912,E2 -27879.912} C_VEL
LIN {X 0,Y 157.972,Z 804.316,A -85,B 0,C 180,E1 -27881.746,E2 -27881.746} C_VEL
LIN {X 0,Y 167.575,Z 793.015,A -85,B 0,C 180,E1 -27883.606,E2 -27883.606} C_VEL
LIN {X 0,Y 175.584,Z 782.461,A -85,B 0,C 180,E1 -27884.931,E2 -27884.931} C_VEL
LIN {X 0,Y 182.867,Z 771.66,A -85,B 0,C 180,E1 -27886.023,E2 -27886.023} C_VEL
LIN {X 0,Y 189.886,Z 759.859,A -85,B 0,C 180,E1 -27886.964,E2 -27886.964} C_VEL
LIN {X 0,Y 195.975,Z 748.086,A -85,B 0,C 180,E1 -27887.743,E2 -27887.743} C_VEL
LIN {X 0,Y 201.355,Z 736.08,A -85,B 0,C 180,E1 -27888.366,E2 -27888.366} C_VEL
LIN {X 0,Y 206.345,Z 722.884,A -85,B 0,C 180,E1 -27888.906,E2 -27888.906} C_VEL
LIN {X 0,Y 206.782,Z 721.6,A -85,B 0,C 180,E1 -27888.948,E2 -27888.948} C_VEL
LIN {X 0,Y 207.907,Z 717.924,A -85,B 0,C 180,E1 -27889.257,E2 -27889.257} C_VEL
LIN {X 0,Y 209.061,Z 712.254,A -85,B 0,C 180,E1 -27890.228,E2 -27890.228} C_VEL
LIN {X 0,Y 210.169,Z 706.533,A -85,B 0,C 180,E1 -27891.158,E2 -27891.158} C_VEL
LIN {X 0,Y 211.073,Z 702.784,A -85,B 0,C 180,E1 -27891.42,E2 -27891.42} C_VEL
LIN {X 0,Y 214.48,Z 685.953,A -85,B 0,C 180,E1 -27891.771,E2 -27891.771} C_VEL
LIN {X 0,Y 217.883,Z 659.221,A -85,B 0,C 180,E1 -27892.217,E2 -27892.217} C_VEL
LIN {X 0,Y 219.017,Z 649.321,A -85,B 0,C 180,E1 -27892.394,E2 -27892.394} C_VEL
LIN {X 0,Y 218.424,Z 647.403,A -85,B 0,C 180,E1 -27894.186,E2 -27894.186} C_VEL
LIN {X 0,Y 217.801,Z 645.064,A -85,B 0,C 180,E1 -27897.225,E2 -27897.225} C_VEL
LIN {X 0,Y 217.584,Z 644.436,A -85,B 0,C 180,E1 -27900,E2 -27900} C_VEL
LIN {X 0,Y 217.905,Z 645.415,A -85,B 0,C 180,E1 -27903.858,E2 -27903.858} C_VEL
LIN {X 0,Y 218.749,Z 648.526,A -85,B 0,C 180,E1 -27907.289,E2 -27907.289} C_VEL
LIN {X 0,Y 220.131,Z 652.861,A -85,B 0,C 180,E1 -27910.559,E2 -27910.559} C_VEL
LIN {X 0,Y 221.699,Z 658.378,A -85,B 0,C 180,E1 -27913.374,E2 -27913.374} C_VEL
LIN {X 0,Y 227.354,Z 675.171,A -85,B 0,C 180,E1 -27920.147,E2 -27920.147} C_VEL
LIN {X 0,Y 232.512,Z 685.126,A -85,B 0,C 180,E1 -27924.379,E2 -27924.379} C_VEL
LIN {X 0,Y 238.602,Z 694.297,A -85,B 0,C 180,E1 -27928.476,E2 -27928.476} C_VEL
LIN {X 0,Y 249.879,Z 707.184,A -85,B 0,C 180,E1 -27934.473,E2 -27934.473} C_VEL
LIN {X 0,Y 266.633,Z 721.782,A -85,B 0,C 180,E1 -27941.22,E2 -27941.22} C_VEL
LIN {X 0,Y 274.211,Z 727.572,A -85,B 0,C 180,E1 -27943.788,E2 -27943.788} C_VEL
LIN {X 0,Y 281.531,Z 733.335,A -85,B 0,C 180,E1 -27946.38,E2 -27946.38} C_VEL
LIN {X 0,Y 288.579,Z 738.849,A -85,B 0,C 180,E1 -27949.022,E2 -27949.022} C_VEL
LIN {X 0,Y 295.864,Z 744.269,A -85,B 0,C 180,E1 -27951.859,E2 -27951.859} C_VEL
LIN {X 0,Y 302.093,Z 749.195,A -85,B 0,C 180,E1 -27954.512,E2 -27954.512} C_VEL
LIN {X 0,Y 307.075,Z 752.787,A -85,B 0,C 180,E1 -27956.683,E2 -27956.683} C_VEL
LIN {X 0,Y 313.384,Z 757.786,A -85,B 0,C 180,E1 -27959.679,E2 -27959.679} C_VEL
LIN {X 0,Y 318.841,Z 761.549,A -85,B 0,C 180,E1 -27962.427,E2 -27962.427} C_VEL
LIN {X 0,Y 321.927,Z 763.99,A -85,B 0,C 180,E1 -27964.112,E2 -27964.112} C_VEL
LIN {X 0,Y 327.438,Z 767.847,A -85,B 0,C 180,E1 -27967.357,E2 -27967.357} C_VEL
LIN {X 0,Y 330.54,Z 769.77,A -85,B 0,C 180,E1 -27969.313,E2 -27969.313} C_VEL
LIN {X 0,Y 333.58,Z 772.14,A -85,B 0,C 180,E1 -27971.578,E2 -27971.578} C_VEL
LIN {X 0,Y 336.768,Z 774.65,A -85,B 0,C 180,E1 -27974.259,E2 -27974.259} C_VEL
LIN {X 0,Y 339.514,Z 776.507,A -85,B 0,C 180,E1 -27976.839,E2 -27976.839} C_VEL
LIN {X 0,Y 341.838,Z 777.66,A -85,B 0,C 180,E1 -27979.337,E2 -27979.337} C_VEL
LIN {X 0,Y 343.692,Z 778.478,A -85,B 0,C 180,E1 -27981.771,E2 -27981.771} C_VEL
LIN {X 0,Y 345.004,Z 779.184,A -85,B 0,C 180,E1 -27984.154,E2 -27984.154} C_VEL
LIN {X 0,Y 345.898,Z 779.632,A -85,B 0,C 180,E1 -27986.505,E2 -27986.505} C_VEL
LIN {X 0,Y 346.411,Z 779.758,A -85,B 0,C 180,E1 -27988.838,E2 -27988.838} C_VEL
LIN {X 0,Y 346.388,Z 779.745,A -85,B 0,C 180,E1 -27991.163,E2 -27991.163} C_VEL
LIN {X 0,Y 345.873,Z 779.646,A -85,B 0,C 180,E1 -27993.495,E2 -27993.495} C_VEL
LIN {X 0,Y 345.016,Z 779.175,A -85,B 0,C 180,E1 -27995.846,E2 -27995.846} C_VEL
LIN {X 0,Y 343.711,Z 778.493,A -85,B 0,C 180,E1 -27998.229,E2 -27998.229} C_VEL
LIN {X 0,Y 341.834,Z 777.689,A -85,B 0,C 180,E1 -28000.663,E2 -28000.663} C_VEL
LIN {X 0,Y 339.413,Z 776.397,A -85,B 0,C 180,E1 -28003.298,E2 -28003.298} C_VEL
LIN {X 0,Y 336.402,Z 774.405,A -85,B 0,C 180,E1 -28006.053,E2 -28006.053} C_VEL
LIN {X 0,Y 333.492,Z 772.037,A -85,B 0,C 180,E1 -28008.501,E2 -28008.501} C_VEL
LIN {X 0,Y 330.547,Z 769.783,A -85,B 0,C 180,E1 -28010.69,E2 -28010.69} C_VEL
LIN {X 0,Y 327.247,Z 767.773,A -85,B 0,C 180,E1 -28012.741,E2 -28012.741} C_VEL
LIN {X 0,Y 324.308,Z 765.79,A -85,B 0,C 180,E1 -28014.473,E2 -28014.473} C_VEL
LIN {X 0,Y 321.289,Z 763.475,A -85,B 0,C 180,E1 -28016.254,E2 -28016.254} C_VEL
LIN {X 0,Y 318.157,Z 761.076,A -85,B 0,C 180,E1 -28017.923,E2 -28017.923} C_VEL
LIN {X 0,Y 313.379,Z 757.756,A -85,B 0,C 180,E1 -28020.317,E2 -28020.317} C_VEL
LIN {X 0,Y 307.043,Z 752.837,A -85,B 0,C 180,E1 -28023.321,E2 -28023.321} C_VEL
LIN {X 0,Y 301.863,Z 748.986,A -85,B 0,C 180,E1 -28025.594,E2 -28025.594} C_VEL
LIN {X 0,Y 295.501,Z 743.971,A -85,B 0,C 180,E1 -28028.294,E2 -28028.294} C_VEL
LIN {X 0,Y 287.961,Z 738.341,A -85,B 0,C 180,E1 -28031.22,E2 -28031.22} C_VEL
LIN {X 0,Y 281.553,Z 733.289,A -85,B 0,C 180,E1 -28033.625,E2 -28033.625} C_VEL
LIN {X 0,Y 274.209,Z 727.544,A -85,B 0,C 180,E1 -28036.211,E2 -28036.211} C_VEL
LIN {X 0,Y 259.436,Z 715.849,A -85,B 0,C 180,E1 -28041.461,E2 -28041.461} C_VEL
LIN {X 0,Y 247.406,Z 704.5,A -85,B 0,C 180,E1 -28046.729,E2 -28046.729} C_VEL
LIN {X 0,Y 239.83,Z 695.793,A -85,B 0,C 180,E1 -28050.792,E2 -28050.792} C_VEL
LIN {X 0,Y 233.985,Z 687.605,A -85,B 0,C 180,E1 -28054.539,E2 -28054.539} C_VEL
LIN {X 0,Y 228.268,Z 677.18,A -85,B 0,C 180,E1 -28059.028,E2 -28059.028} C_VEL
LIN {X 0,Y 223.186,Z 663.859,A -85,B 0,C 180,E1 -28064.417,E2 -28064.417} C_VEL
LIN {X 0,Y 221.374,Z 657.202,A -85,B 0,C 180,E1 -28067.16,E2 -28067.16} C_VEL
LIN {X 0,Y 220.009,Z 652.516,A -85,B 0,C 180,E1 -28069.679,E2 -28069.679} C_VEL
LIN {X 0,Y 218.671,Z 648.212,A -85,B 0,C 180,E1 -28072.962,E2 -28072.962} C_VEL
LIN {X 0,Y 217.888,Z 645.244,A -85,B 0,C 180,E1 -28076.302,E2 -28076.302} C_VEL
LIN {X 0,Y 217.581,Z 644.462,A -85,B 0,C 180,E1 -28080,E2 -28080} C_VEL
LIN {X 0,Y 217.906,Z 645.452,A -85,B 0,C 180,E1 -28083.467,E2 -28083.467} C_VEL
LIN {X 0,Y 218.792,Z 648.618,A -85,B 0,C 180,E1 -28086.987,E2 -28086.987} C_VEL
LIN {X 0,Y 219.015,Z 649.34,A -85,B 0,C 180,E1 -28087.607,E2 -28087.607} C_VEL
LIN {X 0,Y 214.696,Z 684.703,A -85,B 0,C 180,E1 -28088.219,E2 -28088.219} C_VEL
LIN {X 0,Y 211.014,Z 703.045,A -85,B 0,C 180,E1 -28088.605,E2 -28088.605} C_VEL
LIN {X 0,Y 206.357,Z 718.972,A -85,B 0,C 180,E1 -28089.017,E2 -28089.017} C_VEL
LIN {X 0,Y 201.718,Z 731.768,A -85,B 0,C 180,E1 -28089.458,E2 -28089.458} C_VEL
LIN {X 0,Y 196.261,Z 744.395,A -85,B 0,C 180,E1 -28090.023,E2 -28090.023} C_VEL
LIN {X 0,Y 190.46,Z 755.945,A -85,B 0,C 180,E1 -28090.676,E2 -28090.676} C_VEL
LIN {X 0,Y 182.946,Z 768.844,A -85,B 0,C 180,E1 -28091.599,E2 -28091.599} C_VEL
LIN {X 0,Y 176.329,Z 778.822,A -85,B 0,C 180,E1 -28092.451,E2 -28092.451} C_VEL
LIN {X 0,Y 168.15,Z 789.789,A -85,B 0,C 180,E1 -28093.655,E2 -28093.655} C_VEL
LIN {X 0,Y 160.055,Z 799.469,A -85,B 0,C 180,E1 -28094.984,E2 -28094.984} C_VEL
LIN {X 0,Y 150.516,Z 809.67,A -85,B 0,C 180,E1 -28096.828,E2 -28096.828} C_VEL
LIN {X 0,Y 141.077,Z 818.616,A -85,B 0,C 180,E1 -28098.828,E2 -28098.828} C_VEL
LIN {X 0,Y 131.894,Z 826.501,A -85,B 0,C 180,E1 -28101.177,E2 -28101.177} C_VEL
LIN {X 0,Y 122.978,Z 833.463,A -85,B 0,C 180,E1 -28103.886,E2 -28103.886} C_VEL
LIN {X 0,Y 114.451,Z 839.606,A -85,B 0,C 180,E1 -28107.08,E2 -28107.08} C_VEL
LIN {X 0,Y 103.583,Z 846.553,A -85,B 0,C 180,E1 -28111.995,E2 -28111.995} C_VEL
LIN {X 0,Y 93.689,Z 852.318,A -85,B 0,C 180,E1 -28118.035,E2 -28118.035} C_VEL
LIN {X 0,Y 87.064,Z 855.942,A -85,B 0,C 180,E1 -28123.408,E2 -28123.408} C_VEL
LIN {X 0,Y 79.647,Z 859.815,A -85,B 0,C 180,E1 -28131.855,E2 -28131.855} C_VEL
LIN {X 0,Y 74.033,Z 862.69,A -85,B 0,C 180,E1 -28141.664,E2 -28141.664} C_VEL
LIN {X 0,Y 70.587,Z 864.604,A -85,B 0,C 180,E1 -28152.621,E2 -28152.621} C_VEL
LIN {X 0,Y 69.777,Z 865.297,A -85,B 0,C 180,E1 -28158.379,E2 -28158.379} C_VEL
LIN {X 0,Y 69.664,Z 865.799,A -85,B 0,C 180,E1 -28170,E2 -28170} C_VEL
LIN {X 0,Y 69.744,Z 865.296,A -85,B 0,C 180,E1 -28181.627,E2 -28181.627} C_VEL
LIN {X 0,Y 71.977,Z 863.839,A -85,B 0,C 180,E1 -28192.989,E2 -28192.989} C_VEL
LIN {X 0,Y 78.251,Z 860.533,A -85,B 0,C 180,E1 -28206.067,E2 -28206.067} C_VEL
LIN {X 0,Y 85.059,Z 856.987,A -85,B 0,C 180,E1 -28214.612,E2 -28214.612} C_VEL
LIN {X 0,Y 91.411,Z 853.608,A -85,B 0,C 180,E1 -28220.248,E2 -28220.248} C_VEL
LIN {X 0,Y 101.007,Z 848.098,A -85,B 0,C 180,E1 -28226.608,E2 -28226.608} C_VEL
LIN {X 0,Y 108.918,Z 843.238,A -85,B 0,C 180,E1 -28230.584,E2 -28230.584} C_VEL
LIN {X 0,Y 120.109,Z 835.57,A -85,B 0,C 180,E1 -28235.085,E2 -28235.085} C_VEL
LIN {X 0,Y 128.893,Z 828.917,A -85,B 0,C 180,E1 -28237.959,E2 -28237.959} C_VEL
LIN {X 0,Y 137.976,Z 821.37,A -85,B 0,C 180,E1 -28240.442,E2 -28240.442} C_VEL
LIN {X 0,Y 147.355,Z 812.799,A -85,B 0,C 180,E1 -28242.528,E2 -28242.528} C_VEL
LIN {X 0,Y 156.499,Z 803.409,A -85,B 0,C 180,E1 -28244.368,E2 -28244.368} C_VEL
LIN {X 0,Y 165.709,Z 792.805,A -85,B 0,C 180,E1 -28245.965,E2 -28245.965} C_VEL
LIN {X 0,Y 173.86,Z 782.249,A -85,B 0,C 180,E1 -28247.211,E2 -28247.211} C_VEL
LIN {X 0,Y 181.279,Z 771.45,A -85,B 0,C 180,E1 -28248.207,E2 -28248.207} C_VEL
LIN {X 0,Y 188.116,Z 760.172,A -85,B 0,C 180,E1 -28249.042,E2 -28249.042} C_VEL
LIN {X 0,Y 194.588,Z 747.875,A -85,B 0,C 180,E1 -28249.793,E2 -28249.793} C_VEL
LIN {X 0,Y 200.043,Z 735.87,A -85,B 0,C 180,E1 -28250.361,E2 -28250.361} C_VEL
LIN {X 0,Y 204.674,Z 723.908,A -85,B 0,C 180,E1 -28250.816,E2 -28250.816} C_VEL
LIN {X 0,Y 208.9,Z 710.704,A -85,B 0,C 180,E1 -28251.204,E2 -28251.204} C_VEL
LIN {X 0,Y 211.073,Z 702.784,A -85,B 0,C 180,E1 -28251.42,E2 -28251.42} C_VEL
LIN {X 0,Y 212.372,Z 697.121,A -85,B 0,C 180,E1 -28251.71,E2 -28251.71} C_VEL
LIN {X 0,Y 213.758,Z 687.958,A -85,B 0,C 180,E1 -28252.672,E2 -28252.672} C_VEL
LIN {X 0,Y 214.762,Z 678.708,A -85,B 0,C 180,E1 -28253.608,E2 -28253.608} C_VEL
LIN {X 0,Y 215.409,Z 672.905,A -85,B 0,C 180,E1 -28253.858,E2 -28253.858} C_VEL
LIN {X 0,Y 217.552,Z 654.57,A -85,B 0,C 180,E1 -28254.153,E2 -28254.153} C_VEL
LIN {X 0,Y 216.932,Z 652.15,A -85,B 0,C 180,E1 -28257.214,E2 -28257.214} C_VEL
LIN {X 0,Y 216.719,Z 651.483,A -85,B 0,C 180,E1 -28260,E2 -28260} C_VEL
LIN {X 0,Y 216.982,Z 652.421,A -85,B 0,C 180,E1 -28263.598,E2 -28263.598} C_VEL
LIN {X 0,Y 217.718,Z 655.397,A -85,B 0,C 180,E1 -28266.894,E2 -28266.894} C_VEL
LIN {X 0,Y 219.051,Z 659.976,A -85,B 0,C 180,E1 -28270.28,E2 -28270.28} C_VEL
LIN {X 0,Y 220.633,Z 666.257,A -85,B 0,C 180,E1 -28273.293,E2 -28273.293} C_VEL
LIN {X 0,Y 225.055,Z 680.715,A -85,B 0,C 180,E1 -28279.14,E2 -28279.14} C_VEL
LIN {X 0,Y 229.74,Z 690.768,A -85,B 0,C 180,E1 -28283.519,E2 -28283.519} C_VEL
LIN {X 0,Y 235.809,Z 700.483,A -85,B 0,C 180,E1 -28287.995,E2 -28287.995} C_VEL
LIN {X 0,Y 247.501,Z 714.212,A -85,B 0,C 180,E1 -28294.604,E2 -28294.604} C_VEL
LIN {X 0,Y 264.427,Z 728.955,A -85,B 0,C 180,E1 -28301.64,E2 -28301.64} C_VEL
LIN {X 0,Y 273.307,Z 735.916,A -85,B 0,C 180,E1 -28304.76,E2 -28304.76} C_VEL
LIN {X 0,Y 281.046,Z 741.794,A -85,B 0,C 180,E1 -28307.533,E2 -28307.533} C_VEL
LIN {X 0,Y 288.033,Z 747.301,A -85,B 0,C 180,E1 -28310.227,E2 -28310.227} C_VEL
LIN {X 0,Y 293.188,Z 751.177,A -85,B 0,C 180,E1 -28312.282,E2 -28312.282} C_VEL
LIN {X 0,Y 299.88,Z 756.315,A -85,B 0,C 180,E1 -28315.11,E2 -28315.11} C_VEL
LIN {X 0,Y 304.826,Z 760.045,A -85,B 0,C 180,E1 -28317.332,E2 -28317.332} C_VEL
LIN {X 0,Y 310.641,Z 764.517,A -85,B 0,C 180,E1 -28320.151,E2 -28320.151} C_VEL
LIN {X 0,Y 314.339,Z 767.068,A -85,B 0,C 180,E1 -28321.998,E2 -28321.998} C_VEL
LIN {X 0,Y 317.593,Z 769.533,A -85,B 0,C 180,E1 -28323.732,E2 -28323.732} C_VEL
LIN {X 0,Y 323.111,Z 773.506,A -85,B 0,C 180,E1 -28326.952,E2 -28326.952} C_VEL
LIN {X 0,Y 325.624,Z 775.034,A -85,B 0,C 180,E1 -28328.475,E2 -28328.475} C_VEL
LIN {X 0,Y 328.363,Z 776.893,A -85,B 0,C 180,E1 -28330.344,E2 -28330.344} C_VEL
LIN {X 0,Y 331.349,Z 779.361,A -85,B 0,C 180,E1 -28332.726,E2 -28332.726} C_VEL
LIN {X 0,Y 334.39,Z 781.615,A -85,B 0,C 180,E1 -28335.392,E2 -28335.392} C_VEL
LIN {X 0,Y 337.27,Z 783.372,A -85,B 0,C 180,E1 -28338.341,E2 -28338.341} C_VEL
LIN {X 0,Y 339.135,Z 784.134,A -85,B 0,C 180,E1 -28340.457,E2 -28340.457} C_VEL
LIN {X 0,Y 340.797,Z 784.888,A -85,B 0,C 180,E1 -28342.893,E2 -28342.893} C_VEL
LIN {X 0,Y 341.877,Z 785.577,A -85,B 0,C 180,E1 -28345.283,E2 -28345.283} C_VEL
LIN {X 0,Y 342.675,Z 785.779,A -85,B 0,C 180,E1 -28347.649,E2 -28347.649} C_VEL
LIN {X 0,Y 342.83,Z 785.985,A -85,B 0,C 180,E1 -28350,E2 -28350} C_VEL
LIN {X 0,Y 342.634,Z 785.8,A -85,B 0,C 180,E1 -28352.351,E2 -28352.351} C_VEL
LIN {X 0,Y 341.92,Z 785.517,A -85,B 0,C 180,E1 -28354.716,E2 -28354.716} C_VEL
LIN {X 0,Y 340.803,Z 784.923,A -85,B 0,C 180,E1 -28357.107,E2 -28357.107} C_VEL
LIN {X 0,Y 339.108,Z 784.201,A -85,B 0,C 180,E1 -28359.543,E2 -28359.543} C_VEL
LIN {X 0,Y 336.933,Z 783.153,A -85,B 0,C 180,E1 -28362.039,E2 -28362.039} C_VEL
LIN {X 0,Y 334.263,Z 781.531,A -85,B 0,C 180,E1 -28364.725,E2 -28364.725} C_VEL
LIN {X 0,Y 331.286,Z 779.344,A -85,B 0,C 180,E1 -28367.325,E2 -28367.325} C_VEL
LIN {X 0,Y 327.806,Z 776.462,A -85,B 0,C 180,E1 -28370.061,E2 -28370.061} C_VEL
LIN {X 0,Y 325.298,Z 774.856,A -85,B 0,C 180,E1 -28371.721,E2 -28371.721} C_VEL
LIN {X 0,Y 320.417,Z 771.704,A -85,B 0,C 180,E1 -28374.629,E2 -28374.629} C_VEL
LIN {X 0,Y 315.953,Z 768.254,A -85,B 0,C 180,E1 -28377.159,E2 -28377.159} C_VEL
LIN {X 0,Y 310.688,Z 764.476,A -85,B 0,C 180,E1 -28379.844,E2 -28379.844} C_VEL
LIN {X 0,Y 306.359,Z 761.328,A -85,B 0,C 180,E1 -28381.92,E2 -28381.92} C_VEL
LIN {X 0,Y 302.003,Z 757.846,A -85,B 0,C 180,E1 -28383.952,E2 -28383.952} C_VEL
LIN {X 0,Y 296.447,Z 753.744,A -85,B 0,C 180,E1 -28386.347,E2 -28386.347} C_VEL
LIN {X 0,Y 289.797,Z 748.587,A -85,B 0,C 180,E1 -28389.101,E2 -28389.101} C_VEL
LIN {X 0,Y 282.81,Z 743.208,A -85,B 0,C 180,E1 -28391.797,E2 -28391.797} C_VEL
LIN {X 0,Y 275.6,Z 737.68,A -85,B 0,C 180,E1 -28394.438,E2 -28394.438} C_VEL
LIN {X 0,Y 268.146,Z 731.757,A -85,B 0,C 180,E1 -28397.044,E2 -28397.044} C_VEL
LIN {X 0,Y 250.671,Z 717.141,A -85,B 0,C 180,E1 -28403.931,E2 -28403.931} C_VEL
LIN {X 0,Y 238.378,Z 703.972,A -85,B 0,C 180,E1 -28410.347,E2 -28410.347} C_VEL
LIN {X 0,Y 231.274,Z 693.523,A -85,B 0,C 180,E1 -28415.243,E2 -28415.243} C_VEL
LIN {X 0,Y 226.05,Z 682.984,A -85,B 0,C 180,E1 -28419.893,E2 -28419.893} C_VEL
LIN {X 0,Y 221.55,Z 669.995,A -85,B 0,C 180,E1 -28425.242,E2 -28425.242} C_VEL
LIN {X 0,Y 219.878,Z 663.291,A -85,B 0,C 180,E1 -28428.038,E2 -28428.038} C_VEL
LIN {X 0,Y 218.72,Z 658.956,A -85,B 0,C 180,E1 -28430.42,E2 -28430.42} C_VEL
LIN {X 0,Y 217.573,Z 654.772,A -85,B 0,C 180,E1 -28433.625,E2 -28433.625} C_VEL
LIN {X 0,Y 216.94,Z 652.157,A -85,B 0,C 180,E1 -28436.75,E2 -28436.75} C_VEL
LIN {X 0,Y 216.716,Z 651.614,A -85,B 0,C 180,E1 -28440.465,E2 -28440.465} C_VEL
LIN {X 0,Y 216.98,Z 652.353,A -85,B 0,C 180,E1 -28443.134,E2 -28443.134} C_VEL
LIN {X 0,Y 217.546,Z 654.634,A -85,B 0,C 180,E1 -28445.85,E2 -28445.85} C_VEL
LIN {X 0,Y 213.734,Z 684.891,A -85,B 0,C 180,E1 -28446.339,E2 -28446.339} C_VEL
LIN {X 0,Y 209.759,Z 703.931,A -85,B 0,C 180,E1 -28446.706,E2 -28446.706} C_VEL
LIN {X 0,Y 205.36,Z 718.761,A -85,B 0,C 180,E1 -28447.051,E2 -28447.051} C_VEL
LIN {X 0,Y 200.67,Z 731.558,A -85,B 0,C 180,E1 -28447.452,E2 -28447.452} C_VEL
LIN {X 0,Y 195.147,Z 744.184,A -85,B 0,C 180,E1 -28447.962,E2 -28447.962} C_VEL
LIN {X 0,Y 188.71,Z 756.726,A -85,B 0,C 180,E1 -28448.611,E2 -28448.611} C_VEL
LIN {X 0,Y 181.646,Z 768.633,A -85,B 0,C 180,E1 -28449.395,E2 -28449.395} C_VEL
LIN {X 0,Y 174.922,Z 778.61,A -85,B 0,C 180,E1 -28450.155,E2 -28450.155} C_VEL
LIN {X 0,Y 166.597,Z 789.576,A -85,B 0,C 180,E1 -28451.249,E2 -28451.249} C_VEL
LIN {X 0,Y 158.354,Z 799.257,A -85,B 0,C 180,E1 -28452.48,E2 -28452.48} C_VEL
LIN {X 0,Y 150.214,Z 807.893,A -85,B 0,C 180,E1 -28453.881,E2 -28453.881} C_VEL
LIN {X 0,Y 138.922,Z 818.403,A -85,B 0,C 180,E1 -28456.017,E2 -28456.017} C_VEL
LIN {X 0,Y 129.465,Z 826.288,A -85,B 0,C 180,E1 -28458.202,E2 -28458.202} C_VEL
LIN {X 0,Y 120.238,Z 833.25,A -85,B 0,C 180,E1 -28460.742,E2 -28460.742} C_VEL
LIN {X 0,Y 111.346,Z 839.392,A -85,B 0,C 180,E1 -28463.766,E2 -28463.766} C_VEL
LIN {X 0,Y 99.943,Z 846.339,A -85,B 0,C 180,E1 -28468.48,E2 -28468.48} C_VEL
LIN {X 0,Y 91.959,Z 850.816,A -85,B 0,C 180,E1 -28472.791,E2 -28472.791} C_VEL
LIN {X 0,Y 82.264,Z 855.728,A -85,B 0,C 180,E1 -28479.747,E2 -28479.747} C_VEL
LIN {X 0,Y 74.095,Z 859.601,A -85,B 0,C 180,E1 -28488.399,E2 -28488.399} C_VEL
LIN {X 0,Y 67.78,Z 862.477,A -85,B 0,C 180,E1 -28498.773,E2 -28498.773} C_VEL
LIN {X 0,Y 63.783,Z 864.392,A -85,B 0,C 180,E1 -28510.698,E2 -28510.698} C_VEL
LIN {X 0,Y 62.795,Z 865.086,A -85,B 0,C 180,E1 -28517.066,E2 -28517.066} C_VEL
LIN {X 0,Y 62.552,Z 865.589,A -85,B 0,C 180,E1 -28530,E2 -28530} C_VEL
LIN {X 0,Y 62.769,Z 865.085,A -85,B 0,C 180,E1 -28542.94,E2 -28542.94} C_VEL
LIN {X 0,Y 65.438,Z 863.627,A -85,B 0,C 180,E1 -28555.441,E2 -28555.441} C_VEL
LIN {X 0,Y 72.035,Z 860.558,A -85,B 0,C 180,E1 -28568.691,E2 -28568.691} C_VEL
LIN {X 0,Y 80.072,Z 856.773,A -85,B 0,C 180,E1 -28578.248,E2 -28578.248} C_VEL
LIN {X 0,Y 86.971,Z 853.395,A -85,B 0,C 180,E1 -28583.908,E2 -28583.908} C_VEL
LIN {X 0,Y 97.221,Z 847.885,A -85,B 0,C 180,E1 -28590.163,E2 -28590.163} C_VEL
LIN {X 0,Y 105.561,Z 843.025,A -85,B 0,C 180,E1 -28593.997,E2 -28593.997} C_VEL
LIN {X 0,Y 117.242,Z 835.356,A -85,B 0,C 180,E1 -28598.298,E2 -28598.298} C_VEL
LIN {X 0,Y 126.365,Z 828.704,A -85,B 0,C 180,E1 -28600.989,E2 -28600.989} C_VEL
LIN {X 0,Y 135.736,Z 821.158,A -85,B 0,C 180,E1 -28603.305,E2 -28603.305} C_VEL
LIN {X 0,Y 145.361,Z 812.587,A -85,B 0,C 180,E1 -28605.228,E2 -28605.228} C_VEL
LIN {X 0,Y 153.97,Z 804.008,A -85,B 0,C 180,E1 -28606.807,E2 -28606.807} C_VEL
LIN {X 0,Y 163.291,Z 793.599,A -85,B 0,C 180,E1 -28608.273,E2 -28608.273} C_VEL
LIN {X 0,Y 171.582,Z 783.18,A -85,B 0,C 180,E1 -28609.425,E2 -28609.425} C_VEL
LIN {X 0,Y 179.959,Z 771.24,A -85,B 0,C 180,E1 -28610.426,E2 -28610.426} C_VEL
LIN {X 0,Y 186.603,Z 760.471,A -85,B 0,C 180,E1 -28611.162,E2 -28611.162} C_VEL
LIN {X 0,Y 192.608,Z 749.406,A -85,B 0,C 180,E1 -28611.782,E2 -28611.782} C_VEL
LIN {X 0,Y 198.547,Z 736.684,A -85,B 0,C 180,E1 -28612.348,E2 -28612.348} C_VEL
LIN {X 0,Y 203.662,Z 723.698,A -85,B 0,C 180,E1 -28612.787,E2 -28612.787} C_VEL
LIN {X 0,Y 208.086,Z 709.93,A -85,B 0,C 180,E1 -28613.158,E2 -28613.158} C_VEL
LIN {X 0,Y 211.38,Z 696.958,A -85,B 0,C 180,E1 -28613.434,E2 -28613.434} C_VEL
LIN {X 0,Y 213.886,Z 683.693,A -85,B 0,C 180,E1 -28613.687,E2 -28613.687} C_VEL
LIN {X 0,Y 215.409,Z 672.905,A -85,B 0,C 180,E1 -28613.858,E2 -28613.858} C_VEL
LIN {X 0,Y 215.736,Z 669.557,A -85,B 0,C 180,E1 -28614.067,E2 -28614.067} C_VEL
LIN {X 0,Y 215.926,Z 666.541,A -85,B 0,C 180,E1 -28614.537,E2 -28614.537} C_VEL
LIN {X 0,Y 216.027,Z 663.497,A -85,B 0,C 180,E1 -28615.323,E2 -28615.323} C_VEL
LIN {X 0,Y 216.035,Z 660.439,A -85,B 0,C 180,E1 -28616.648,E2 -28616.648} C_VEL
LIN {X 0,Y 215.954,Z 659.067,A -85,B 0,C 180,E1 -28617.95,E2 -28617.95} C_VEL
LIN {X 0,Y 215.935,Z 658.997,A -85,B 0,C 180,E1 -28618.143,E2 -28618.143} C_VEL
LIN {X 0,Y 215.852,Z 658.543,A -85,B 0,C 180,E1 -28620,E2 -28620} C_VEL
LIN {X 0,Y 216.056,Z 659.371,A -85,B 0,C 180,E1 -28623.263,E2 -28623.263} C_VEL
LIN {X 0,Y 216.668,Z 662.185,A -85,B 0,C 180,E1 -28626.401,E2 -28626.401} C_VEL
LIN {X 0,Y 217.804,Z 666.523,A -85,B 0,C 180,E1 -28629.622,E2 -28629.622} C_VEL
LIN {X 0,Y 219.126,Z 672.407,A -85,B 0,C 180,E1 -28632.444,E2 -28632.444} C_VEL
LIN {X 0,Y 223.02,Z 686.931,A -85,B 0,C 180,E1 -28638.433,E2 -28638.433} C_VEL
LIN {X 0,Y 227.46,Z 697.438,A -85,B 0,C 180,E1 -28643.153,E2 -28643.153} C_VEL
LIN {X 0,Y 232.752,Z 706.542,A -85,B 0,C 180,E1 -28647.478,E2 -28647.478} C_VEL
LIN {X 0,Y 242.382,Z 718.489,A -85,B 0,C 180,E1 -28653.429,E2 -28653.429} C_VEL
LIN {X 0,Y 257.234,Z 732.181,A -85,B 0,C 180,E1 -28660.267,E2 -28660.267} C_VEL
LIN {X 0,Y 269.412,Z 741.868,A -85,B 0,C 180,E1 -28664.775,E2 -28664.775} C_VEL
LIN {X 0,Y 276.782,Z 747.45,A -85,B 0,C 180,E1 -28667.421,E2 -28667.421} C_VEL
LIN {X 0,Y 283.865,Z 753.032,A -85,B 0,C 180,E1 -28670.13,E2 -28670.13} C_VEL
LIN {X 0,Y 290.362,Z 758.016,A -85,B 0,C 180,E1 -28672.765,E2 -28672.765} C_VEL
LIN {X 0,Y 296.365,Z 762.493,A -85,B 0,C 180,E1 -28675.311,E2 -28675.311} C_VEL
LIN {X 0,Y 301.312,Z 766.313,A -85,B 0,C 180,E1 -28677.557,E2 -28677.557} C_VEL
LIN {X 0,Y 307.205,Z 770.749,A -85,B 0,C 180,E1 -28680.38,E2 -28680.38} C_VEL
LIN {X 0,Y 312.862,Z 774.838,A -85,B 0,C 180,E1 -28683.304,E2 -28683.304} C_VEL
LIN {X 0,Y 318.592,Z 779.018,A -85,B 0,C 180,E1 -28686.605,E2 -28686.605} C_VEL
LIN {X 0,Y 322.976,Z 781.803,A -85,B 0,C 180,E1 -28689.337,E2 -28689.337} C_VEL
LIN {X 0,Y 325.993,Z 784.083,A -85,B 0,C 180,E1 -28691.545,E2 -28691.545} C_VEL
LIN {X 0,Y 328.949,Z 786.475,A -85,B 0,C 180,E1 -28694.031,E2 -28694.031} C_VEL
LIN {X 0,Y 331.943,Z 788.474,A -85,B 0,C 180,E1 -28696.884,E2 -28696.884} C_VEL
LIN {X 0,Y 334.065,Z 789.561,A -85,B 0,C 180,E1 -28699.086,E2 -28699.086} C_VEL
LIN {X 0,Y 336.07,Z 790.461,A -85,B 0,C 180,E1 -28701.583,E2 -28701.583} C_VEL
LIN {X 0,Y 337.47,Z 791.203,A -85,B 0,C 180,E1 -28704.023,E2 -28704.023} C_VEL
LIN {X 0,Y 338.393,Z 791.66,A -85,B 0,C 180,E1 -28706.428,E2 -28706.428} C_VEL
LIN {X 0,Y 338.933,Z 791.797,A -85,B 0,C 180,E1 -28708.812,E2 -28708.812} C_VEL
LIN {X 0,Y 338.901,Z 791.791,A -85,B 0,C 180,E1 -28711.188,E2 -28711.188} C_VEL
LIN {X 0,Y 338.374,Z 791.675,A -85,B 0,C 180,E1 -28713.572,E2 -28713.572} C_VEL
LIN {X 0,Y 337.498,Z 791.198,A -85,B 0,C 180,E1 -28715.976,E2 -28715.976} C_VEL
LIN {X 0,Y 336.081,Z 790.486,A -85,B 0,C 180,E1 -28718.417,E2 -28718.417} C_VEL
LIN {X 0,Y 334.043,Z 789.568,A -85,B 0,C 180,E1 -28720.915,E2 -28720.915} C_VEL
LIN {X 0,Y 331.6,Z 788.207,A -85,B 0,C 180,E1 -28723.481,E2 -28723.481} C_VEL
LIN {X 0,Y 328.757,Z 786.313,A -85,B 0,C 180,E1 -28726.135,E2 -28726.135} C_VEL
LIN {X 0,Y 325.414,Z 783.638,A -85,B 0,C 180,E1 -28728.902,E2 -28728.902} C_VEL
LIN {X 0,Y 322.974,Z 781.799,A -85,B 0,C 180,E1 -28730.662,E2 -28730.662} C_VEL
LIN {X 0,Y 319.847,Z 779.834,A -85,B 0,C 180,E1 -28732.653,E2 -28732.653} C_VEL
LIN {X 0,Y 315.832,Z 777.104,A -85,B 0,C 180,E1 -28735.01,E2 -28735.01} C_VEL
LIN {X 0,Y 310.413,Z 772.959,A -85,B 0,C 180,E1 -28737.996,E2 -28737.996} C_VEL
LIN {X 0,Y 305.568,Z 769.578,A -85,B 0,C 180,E1 -28740.397,E2 -28740.397} C_VEL
LIN {X 0,Y 300.717,Z 765.853,A -85,B 0,C 180,E1 -28742.718,E2 -28742.718} C_VEL
LIN {X 0,Y 296.366,Z 762.513,A -85,B 0,C 180,E1 -28744.689,E2 -28744.689} C_VEL
LIN {X 0,Y 290.361,Z 758.01,A -85,B 0,C 180,E1 -28747.236,E2 -28747.236} C_VEL
LIN {X 0,Y 286.268,Z 754.798,A -85,B 0,C 180,E1 -28748.921,E2 -28748.921} C_VEL
LIN {X 0,Y 278.611,Z 748.885,A -85,B 0,C 180,E1 -28751.904,E2 -28751.904} C_VEL
LIN {X 0,Y 271.451,Z 743.434,A -85,B 0,C 180,E1 -28754.498,E2 -28754.498} C_VEL
LIN {X 0,Y 262.027,Z 736.055,A -85,B 0,C 180,E1 -28757.892,E2 -28757.892} C_VEL
LIN {X 0,Y 244.095,Z 720.282,A -85,B 0,C 180,E1 -28765.682,E2 -28765.682} C_VEL
LIN {X 0,Y 234.091,Z 708.364,A -85,B 0,C 180,E1 -28771.598,E2 -28771.598} C_VEL
LIN {X 0,Y 228.519,Z 699.536,A -85,B 0,C 180,E1 -28775.892,E2 -28775.892} C_VEL
LIN {X 0,Y 223.82,Z 689.151,A -85,B 0,C 180,E1 -28780.601,E2 -28780.601} C_VEL
LIN {X 0,Y 220.618,Z 678.959,A -85,B 0,C 180,E1 -28784.89,E2 -28784.89} C_VEL
LIN {X 0,Y 218.441,Z 669.331,A -85,B 0,C 180,E1 -28788.929,E2 -28788.929} C_VEL
LIN {X 0,Y 217.481,Z 665.412,A -85,B 0,C 180,E1 -28791.141,E2 -28791.141} C_VEL
LIN {X 0,Y 216.531,Z 661.459,A -85,B 0,C 180,E1 -28794.179,E2 -28794.179} C_VEL
LIN {X 0,Y 216.003,Z 659.096,A -85,B 0,C 180,E1 -28797.203,E2 -28797.203} C_VEL
LIN {X 0,Y 215.851,Z 658.555,A -85,B 0,C 180,E1 -28800,E2 -28800} C_VEL
LIN {X 0,Y 216.063,Z 659.425,A -85,B 0,C 180,E1 -28802.914,E2 -28802.914} C_VEL
LIN {X 0,Y 216.228,Z 660.368,A -85,B 0,C 180,E1 -28804.066,E2 -28804.066} C_VEL
LIN {X 0,Y 212.829,Z 686.194,A -85,B 0,C 180,E1 -28804.465,E2 -28804.465} C_VEL
LIN {X 0,Y 208.788,Z 704.646,A -85,B 0,C 180,E1 -28804.788,E2 -28804.788} C_VEL
LIN {X 0,Y 204.61,Z 718.552,A -85,B 0,C 180,E1 -28805.078,E2 -28805.078} C_VEL
LIN {X 0,Y 199.874,Z 731.348,A -85,B 0,C 180,E1 -28805.434,E2 -28805.434} C_VEL
LIN {X 0,Y 194.289,Z 743.974,A -85,B 0,C 180,E1 -28805.883,E2 -28805.883} C_VEL
LIN {X 0,Y 187.9,Z 756.292,A -85,B 0,C 180,E1 -28806.443,E2 -28806.443} C_VEL
LIN {X 0,Y 180.619,Z 768.422,A -85,B 0,C 180,E1 -28807.163,E2 -28807.163} C_VEL
LIN {X 0,Y 173.808,Z 778.4,A -85,B 0,C 180,E1 -28807.843,E2 -28807.843} C_VEL
LIN {X 0,Y 165.351,Z 789.365,A -85,B 0,C 180,E1 -28808.818,E2 -28808.818} C_VEL
LIN {X 0,Y 156.956,Z 799.044,A -85,B 0,C 180,E1 -28809.914,E2 -28809.914} C_VEL
LIN {X 0,Y 148.649,Z 807.68,A -85,B 0,C 180,E1 -28811.182,E2 -28811.182} C_VEL
LIN {X 0,Y 138.762,Z 816.815,A -85,B 0,C 180,E1 -28812.851,E2 -28812.851} C_VEL
LIN {X 0,Y 127.398,Z 826.075,A -85,B 0,C 180,E1 -28815.121,E2 -28815.121} C_VEL
LIN {X 0,Y 117.869,Z 833.036,A -85,B 0,C 180,E1 -28817.448,E2 -28817.448} C_VEL
LIN {X 0,Y 108.631,Z 839.178,A -85,B 0,C 180,E1 -28820.27,E2 -28820.27} C_VEL
LIN {X 0,Y 96.711,Z 846.126,A -85,B 0,C 180,E1 -28824.72,E2 -28824.72} C_VEL
LIN {X 0,Y 88.254,Z 850.602,A -85,B 0,C 180,E1 -28828.843,E2 -28828.843} C_VEL
LIN {X 0,Y 77.842,Z 855.515,A -85,B 0,C 180,E1 -28835.655,E2 -28835.655} C_VEL
LIN {X 0,Y 68.853,Z 859.387,A -85,B 0,C 180,E1 -28844.398,E2 -28844.398} C_VEL
LIN {X 0,Y 61.735,Z 862.265,A -85,B 0,C 180,E1 -28855.306,E2 -28855.306} C_VEL
LIN {X 0,Y 57.051,Z 864.179,A -85,B 0,C 180,E1 -28868.312,E2 -28868.312} C_VEL
LIN {X 0,Y 55.834,Z 864.874,A -85,B 0,C 180,E1 -28875.42,E2 -28875.42} C_VEL
LIN {X 0,Y 55.46,Z 865.379,A -85,B 0,C 180,E1 -28890,E2 -28890} C_VEL
LIN {X 0,Y 55.814,Z 864.873,A -85,B 0,C 180,E1 -28904.586,E2 -28904.586} C_VEL
LIN {X 0,Y 59.049,Z 863.415,A -85,B 0,C 180,E1 -28918.429,E2 -28918.429} C_VEL
LIN {X 0,Y 66.02,Z 860.576,A -85,B 0,C 180,E1 -28931.825,E2 -28931.825} C_VEL
LIN {X 0,Y 75.459,Z 856.56,A -85,B 0,C 180,E1 -28942.339,E2 -28942.339} C_VEL
LIN {X 0,Y 82.909,Z 853.181,A -85,B 0,C 180,E1 -28947.958,E2 -28947.958} C_VEL
LIN {X 0,Y 91.252,Z 849.085,A -85,B 0,C 180,E1 -28952.744,E2 -28952.744} C_VEL
LIN {X 0,Y 102.601,Z 842.811,A -85,B 0,C 180,E1 -28957.624,E2 -28957.624} C_VEL
LIN {X 0,Y 114.767,Z 835.142,A -85,B 0,C 180,E1 -28961.65,E2 -28961.65} C_VEL
LIN {X 0,Y 124.198,Z 828.49,A -85,B 0,C 180,E1 -28964.145,E2 -28964.145} C_VEL
LIN {X 0,Y 133.851,Z 820.945,A -85,B 0,C 180,E1 -28966.249,E2 -28966.249} C_VEL
LIN {X 0,Y 143.696,Z 812.374,A -85,B 0,C 180,E1 -28968.001,E2 -28968.001} C_VEL
LIN {X 0,Y 153.674,Z 802.539,A -85,B 0,C 180,E1 -28969.604,E2 -28969.604} C_VEL
LIN {X 0,Y 162.832,Z 792.382,A -85,B 0,C 180,E1 -28970.854,E2 -28970.854} C_VEL
LIN {X 0,Y 171.258,Z 781.826,A -85,B 0,C 180,E1 -28971.892,E2 -28971.892} C_VEL
LIN {X 0,Y 178.912,Z 771.029,A -85,B 0,C 180,E1 -28972.677,E2 -28972.677} C_VEL
LIN {X 0,Y 186.154,Z 759.355,A -85,B 0,C 180,E1 -28973.391,E2 -28973.391} C_VEL
LIN {X 0,Y 192.574,Z 747.454,A -85,B 0,C 180,E1 -28973.971,E2 -28973.971} C_VEL
LIN {X 0,Y 198.155,Z 735.449,A -85,B 0,C 180,E1 -28974.427,E2 -28974.427} C_VEL
LIN {X 0,Y 203.321,Z 722.254,A -85,B 0,C 180,E1 -28974.815,E2 -28974.815} C_VEL
LIN {X 0,Y 207.46,Z 709.36,A -85,B 0,C 180,E1 -28975.118,E2 -28975.118} C_VEL
LIN {X 0,Y 210.849,Z 696.009,A -85,B 0,C 180,E1 -28975.357,E2 -28975.357} C_VEL
LIN {X 0,Y 213.176,Z 683.79,A -85,B 0,C 180,E1 -28975.578,E2 -28975.578} C_VEL
LIN {X 0,Y 216.228,Z 660.368,A -85,B 0,C 180,E1 -28975.935,E2 -28975.935} C_VEL
LIN {X 0,Y 216.029,Z 659.153,A -85,B 0,C 180,E1 -28977.436,E2 -28977.436} C_VEL
LIN {X 0,Y 215.935,Z 658.997,A -85,B 0,C 180,E1 -28978.143,E2 -28978.143} C_VEL
LIN {X 0,Y 215.814,Z 659.124,A -85,B 0,C 180,E1 -28979.185,E2 -28979.185} C_VEL
LIN {X 0,Y 215.682,Z 659.914,A -85,B 0,C 180,E1 -28980.21,E2 -28980.21} C_VEL
LIN {X 0,Y 215.462,Z 662.759,A -85,B 0,C 180,E1 -28982.187,E2 -28982.187} C_VEL
LIN {X 0,Y 215.496,Z 667.927,A -85,B 0,C 180,E1 -28985.14,E2 -28985.14} C_VEL
LIN {X 0,Y 215.701,Z 669.24,A -85,B 0,C 180,E1 -28986.163,E2 -28986.163} C_VEL
LIN {X 0,Y 216.624,Z 673.31,A -85,B 0,C 180,E1 -28989.07,E2 -28989.07} C_VEL
LIN {X 0,Y 217.496,Z 678.418,A -85,B 0,C 180,E1 -28991.54,E2 -28991.54} C_VEL
LIN {X 0,Y 220.214,Z 691.158,A -85,B 0,C 180,E1 -28996.871,E2 -28996.871} C_VEL
LIN {X 0,Y 224.237,Z 702.474,A -85,B 0,C 180,E1 -29002.031,E2 -29002.031} C_VEL
LIN {X 0,Y 228.963,Z 711.558,A -85,B 0,C 180,E1 -29006.428,E2 -29006.428} C_VEL
LIN {X 0,Y 240.022,Z 725.809,A -85,B 0,C 180,E1 -29013.802,E2 -29013.802} C_VEL
LIN {X 0,Y 255.878,Z 740.181,A -85,B 0,C 180,E1 -29021.237,E2 -29021.237} C_VEL
LIN {X 0,Y 266.758,Z 748.792,A -85,B 0,C 180,E1 -29025.343,E2 -29025.343} C_VEL
LIN {X 0,Y 274.119,Z 754.448,A -85,B 0,C 180,E1 -29028.031,E2 -29028.031} C_VEL
LIN {X 0,Y 279.209,Z 758.398,A -85,B 0,C 180,E1 -29029.982,E2 -29029.982} C_VEL
LIN {X 0,Y 284.724,Z 762.538,A -85,B 0,C 180,E1 -29032.173,E2 -29032.173} C_VEL
LIN {X 0,Y 290.111,Z 766.743,A -85,B 0,C 180,E1 -29034.452,E2 -29034.452} C_VEL
LIN {X 0,Y 295.56,Z 770.762,A -85,B 0,C 180,E1 -29036.846,E2 -29036.846} C_VEL
LIN {X 0,Y 300.033,Z 774.32,A -85,B 0,C 180,E1 -29038.981,E2 -29038.981} C_VEL
LIN {X 0,Y 304.652,Z 777.629,A -85,B 0,C 180,E1 -29041.236,E2 -29041.236} C_VEL
LIN {X 0,Y 307.884,Z 779.978,A -85,B 0,C 180,E1 -29042.903,E2 -29042.903} C_VEL
LIN {X 0,Y 311.028,Z 782.369,A -85,B 0,C 180,E1 -29044.666,E2 -29044.666} C_VEL
LIN {X 0,Y 314.19,Z 784.606,A -85,B 0,C 180,E1 -29046.506,E2 -29046.506} C_VEL
LIN {X 0,Y 317.399,Z 786.603,A -85,B 0,C 180,E1 -29048.43,E2 -29048.43} C_VEL
LIN {X 0,Y 320.844,Z 789.042,A -85,B 0,C 180,E1 -29050.818,E2 -29050.818} C_VEL
LIN {X 0,Y 324.297,Z 791.812,A -85,B 0,C 180,E1 -29053.637,E2 -29053.637} C_VEL
LIN {X 0,Y 327.182,Z 793.859,A -85,B 0,C 180,E1 -29056.333,E2 -29056.333} C_VEL
LIN {X 0,Y 329.744,Z 795.248,A -85,B 0,C 180,E1 -29058.941,E2 -29058.941} C_VEL
LIN {X 0,Y 331.832,Z 796.161,A -85,B 0,C 180,E1 -29061.474,E2 -29061.474} C_VEL
LIN {X 0,Y 333.239,Z 796.898,A -85,B 0,C 180,E1 -29063.947,E2 -29063.947} C_VEL
LIN {X 0,Y 334.2,Z 797.368,A -85,B 0,C 180,E1 -29066.383,E2 -29066.383} C_VEL
LIN {X 0,Y 334.764,Z 797.523,A -85,B 0,C 180,E1 -29068.797,E2 -29068.797} C_VEL
LIN {X 0,Y 334.719,Z 797.53,A -85,B 0,C 180,E1 -29071.203,E2 -29071.203} C_VEL
LIN {X 0,Y 334.177,Z 797.387,A -85,B 0,C 180,E1 -29073.617,E2 -29073.617} C_VEL
LIN {X 0,Y 333.274,Z 796.888,A -85,B 0,C 180,E1 -29076.052,E2 -29076.052} C_VEL
LIN {X 0,Y 331.823,Z 796.198,A -85,B 0,C 180,E1 -29078.526,E2 -29078.526} C_VEL
LIN {X 0,Y 329.582,Z 795.178,A -85,B 0,C 180,E1 -29081.219,E2 -29081.219} C_VEL
LIN {X 0,Y 326.464,Z 793.349,A -85,B 0,C 180,E1 -29084.366,E2 -29084.366} C_VEL
LIN {X 0,Y 323.464,Z 791.204,A -85,B 0,C 180,E1 -29087.062,E2 -29087.062} C_VEL
LIN {X 0,Y 320.48,Z 788.792,A -85,B 0,C 180,E1 -29089.445,E2 -29089.445} C_VEL
LIN {X 0,Y 317.387,Z 786.621,A -85,B 0,C 180,E1 -29091.564,E2 -29091.564} C_VEL
LIN {X 0,Y 313.668,Z 784.296,A -85,B 0,C 180,E1 -29093.784,E2 -29093.784} C_VEL
LIN {X 0,Y 309.696,Z 781.315,A -85,B 0,C 180,E1 -29096.098,E2 -29096.098} C_VEL
LIN {X 0,Y 306.73,Z 779.064,A -85,B 0,C 180,E1 -29097.74,E2 -29097.74} C_VEL
LIN {X 0,Y 301.414,Z 775.308,A -85,B 0,C 180,E1 -29100.378,E2 -29100.378} C_VEL
LIN {X 0,Y 295.556,Z 770.787,A -85,B 0,C 180,E1 -29103.155,E2 -29103.155} C_VEL
LIN {X 0,Y 290.15,Z 766.717,A -85,B 0,C 180,E1 -29105.543,E2 -29105.543} C_VEL
LIN {X 0,Y 283.694,Z 761.678,A -85,B 0,C 180,E1 -29108.266,E2 -29108.266} C_VEL
LIN {X 0,Y 275.931,Z 755.824,A -85,B 0,C 180,E1 -29111.293,E2 -29111.293} C_VEL
LIN {X 0,Y 270.517,Z 751.543,A -85,B 0,C 180,E1 -29113.329,E2 -29113.329} C_VEL
LIN {X 0,Y 259.458,Z 742.934,A -85,B 0,C 180,E1 -29117.377,E2 -29117.377} C_VEL
LIN {X 0,Y 242.946,Z 728.727,A -85,B 0,C 180,E1 -29124.651,E2 -29124.651} C_VEL
LIN {X 0,Y 232.253,Z 716.462,A -85,B 0,C 180,E1 -29131.043,E2 -29131.043} C_VEL
LIN {X 0,Y 225.769,Z 705.845,A -85,B 0,C 180,E1 -29136.373,E2 -29136.373} C_VEL
LIN {X 0,Y 221.433,Z 695.122,A -85,B 0,C 180,E1 -29141.364,E2 -29141.364} C_VEL
LIN {X 0,Y 218.453,Z 683.501,A -85,B 0,C 180,E1 -29146.379,E2 -29146.379} C_VEL
LIN {X 0,Y 217.042,Z 675.575,A -85,B 0,C 180,E1 -29149.742,E2 -29149.742} C_VEL
LIN {X 0,Y 216.246,Z 671.695,A -85,B 0,C 180,E1 -29151.973,E2 -29151.973} C_VEL
LIN {X 0,Y 215.503,Z 668.203,A -85,B 0,C 180,E1 -29154.736,E2 -29154.736} C_VEL
LIN {X 0,Y 215.135,Z 666.174,A -85,B 0,C 180,E1 -29157.192,E2 -29157.192} C_VEL
LIN {X 0,Y 214.984,Z 665.61,A -85,B 0,C 180,E1 -29160,E2 -29160} C_VEL
LIN {X 0,Y 215.118,Z 666.143,A -85,B 0,C 180,E1 -29162.266,E2 -29162.266} C_VEL
LIN {X 0,Y 211.881,Z 688.959,A -85,B 0,C 180,E1 -29162.606,E2 -29162.606} C_VEL
LIN {X 0,Y 207.993,Z 705.579,A -85,B 0,C 180,E1 -29162.863,E2 -29162.863} C_VEL
LIN {X 0,Y 204.104,Z 718.344,A -85,B 0,C 180,E1 -29163.089,E2 -29163.089} C_VEL
LIN {X 0,Y 199.326,Z 731.139,A -85,B 0,C 180,E1 -29163.397,E2 -29163.397} C_VEL
LIN {X 0,Y 193.688,Z 743.763,A -85,B 0,C 180,E1 -29163.787,E2 -29163.787} C_VEL
LIN {X 0,Y 187.633,Z 755.387,A -85,B 0,C 180,E1 -29164.24,E2 -29164.24} C_VEL
LIN {X 0,Y 179.869,Z 768.211,A -85,B 0,C 180,E1 -29164.907,E2 -29164.907} C_VEL
LIN {X 0,Y 172.118,Z 779.331,A -85,B 0,C 180,E1 -29165.577,E2 -29165.577} C_VEL
LIN {X 0,Y 163.551,Z 790.158,A -85,B 0,C 180,E1 -29166.441,E2 -29166.441} C_VEL
LIN {X 0,Y 154.014,Z 800.784,A -85,B 0,C 180,E1 -29167.547,E2 -29167.547} C_VEL
LIN {X 0,Y 145.744,Z 809.033,A -85,B 0,C 180,E1 -29168.691,E2 -29168.691} C_VEL
LIN {X 0,Y 135.665,Z 817.979,A -85,B 0,C 180,E1 -29170.181,E2 -29170.181} C_VEL
LIN {X 0,Y 125.712,Z 825.862,A -85,B 0,C 180,E1 -29171.952,E2 -29171.952} C_VEL
LIN {X 0,Y 114.807,Z 833.541,A -85,B 0,C 180,E1 -29174.31,E2 -29174.31} C_VEL
LIN {X 0,Y 103.191,Z 840.781,A -85,B 0,C 180,E1 -29177.547,E2 -29177.547} C_VEL
LIN {X 0,Y 93.92,Z 845.913,A -85,B 0,C 180,E1 -29180.715,E2 -29180.715} C_VEL
LIN {X 0,Y 84.998,Z 850.388,A -85,B 0,C 180,E1 -29184.563,E2 -29184.563} C_VEL
LIN {X 0,Y 73.871,Z 855.301,A -85,B 0,C 180,E1 -29191.104,E2 -29191.104} C_VEL
LIN {X 0,Y 64.009,Z 859.174,A -85,B 0,C 180,E1 -29199.775,E2 -29199.775} C_VEL
LIN {X 0,Y 55.969,Z 862.052,A -85,B 0,C 180,E1 -29211.109,E2 -29211.109} C_VEL
LIN {X 0,Y 50.448,Z 863.967,A -85,B 0,C 180,E1 -29225.296,E2 -29225.296} C_VEL
LIN {X 0,Y 48.943,Z 864.662,A -85,B 0,C 180,E1 -29233.311,E2 -29233.311} C_VEL
LIN {X 0,Y 48.35,Z 865.169,A -85,B 0,C 180,E1 -29250,E2 -29250} C_VEL
LIN {X 0,Y 48.927,Z 864.662,A -85,B 0,C 180,E1 -29266.695,E2 -29266.695} C_VEL
LIN {X 0,Y 52.834,Z 863.202,A -85,B 0,C 180,E1 -29282.145,E2 -29282.145} C_VEL
LIN {X 0,Y 60.216,Z 860.601,A -85,B 0,C 180,E1 -29295.549,E2 -29295.549} C_VEL
LIN {X 0,Y 71.27,Z 856.346,A -85,B 0,C 180,E1 -29306.948,E2 -29306.948} C_VEL
LIN {X 0,Y 79.306,Z 852.967,A -85,B 0,C 180,E1 -29312.395,E2 -29312.395} C_VEL
LIN {X 0,Y 90.907,Z 847.458,A -85,B 0,C 180,E1 -29318.078,E2 -29318.078} C_VEL
LIN {X 0,Y 100.08,Z 842.598,A -85,B 0,C 180,E1 -29321.441,E2 -29321.441} C_VEL
LIN {X 0,Y 112.71,Z 834.93,A -85,B 0,C 180,E1 -29325.121,E2 -29325.121} C_VEL
LIN {X 0,Y 122.429,Z 828.278,A -85,B 0,C 180,E1 -29327.384,E2 -29327.384} C_VEL
LIN {X 0,Y 132.325,Z 820.733,A -85,B 0,C 180,E1 -29329.277,E2 -29329.277} C_VEL
LIN {X 0,Y 142.38,Z 812.163,A -85,B 0,C 180,E1 -29330.821,E2 -29330.821} C_VEL
LIN {X 0,Y 152.153,Z 802.736,A -85,B 0,C 180,E1 -29332.205,E2 -29332.205} C_VEL
LIN {X 0,Y 161.847,Z 792.17,A -85,B 0,C 180,E1 -29333.362,E2 -29333.362} C_VEL
LIN {X 0,Y 170.398,Z 781.615,A -85,B 0,C 180,E1 -29334.269,E2 -29334.269} C_VEL
LIN {X 0,Y 178.144,Z 770.818,A -85,B 0,C 180,E1 -29334.951,E2 -29334.951} C_VEL
LIN {X 0,Y 185.466,Z 759.143,A -85,B 0,C 180,E1 -29335.592,E2 -29335.592} C_VEL
LIN {X 0,Y 191.955,Z 747.243,A -85,B 0,C 180,E1 -29336.09,E2 -29336.09} C_VEL
LIN {X 0,Y 197.59,Z 735.239,A -85,B 0,C 180,E1 -29336.488,E2 -29336.488} C_VEL
LIN {X 0,Y 202.802,Z 722.046,A -85,B 0,C 180,E1 -29336.818,E2 -29336.818} C_VEL
LIN {X 0,Y 206.981,Z 709.142,A -85,B 0,C 180,E1 -29337.072,E2 -29337.072} C_VEL
LIN {X 0,Y 210.392,Z 695.808,A -85,B 0,C 180,E1 -29337.29,E2 -29337.29} C_VEL
LIN {X 0,Y 212.816,Z 683.122,A -85,B 0,C 180,E1 -29337.496,E2 -29337.496} C_VEL
LIN {X 0,Y 215.118,Z 666.143,A -85,B 0,C 180,E1 -29337.736,E2 -29337.736} C_VEL
LIN {X 0,Y 214.987,Z 665.587,A -85,B 0,C 180,E1 -29340,E2 -29340} C_VEL
LIN {X 0,Y 215.149,Z 666.406,A -85,B 0,C 180,E1 -29343.042,E2 -29343.042} C_VEL
LIN {X 0,Y 215.651,Z 669.018,A -85,B 0,C 180,E1 -29345.962,E2 -29345.962} C_VEL
LIN {X 0,Y 215.701,Z 669.24,A -85,B 0,C 180,E1 -29346.163,E2 -29346.163} C_VEL
LIN {X 0,Y 215.928,Z 670.768,A -85,B 0,C 180,E1 -29347.12,E2 -29347.12} C_VEL
LIN {X 0,Y 216.102,Z 674.298,A -85,B 0,C 180,E1 -29348.384,E2 -29348.384} C_VEL
LIN {X 0,Y 216.197,Z 685.922,A -85,B 0,C 180,E1 -29351.38,E2 -29351.38} C_VEL
LIN {X 0,Y 216.528,Z 689.348,A -85,B 0,C 180,E1 -29352.698,E2 -29352.698} C_VEL
LIN {X 0,Y 218.931,Z 700.957,A -85,B 0,C 180,E1 -29357.816,E2 -29357.816} C_VEL
LIN {X 0,Y 222.049,Z 709.969,A -85,B 0,C 180,E1 -29362.138,E2 -29362.138} C_VEL
LIN {X 0,Y 225.62,Z 717.383,A -85,B 0,C 180,E1 -29365.854,E2 -29365.854} C_VEL
LIN {X 0,Y 234.784,Z 729.98,A -85,B 0,C 180,E1 -29372.602,E2 -29372.602} C_VEL
LIN {X 0,Y 249.774,Z 744.323,A -85,B 0,C 180,E1 -29380.327,E2 -29380.327} C_VEL
LIN {X 0,Y 262.101,Z 754.16,A -85,B 0,C 180,E1 -29385.281,E2 -29385.281} C_VEL
